LIN {X 0,Y 453.558,Z 377.477,A -85,B 0,C 180,E1 -8448.378,E2 -8448.378} C_VEL
LIN {X 0,Y 453.65,Z 377.467,A -85,B 0,C 180,E1 -8451.985,E2 -8451.985} C_VEL
LIN {X 0,Y 453.669,Z 377.47,A -85,B 0,C 180,E1 -8454.666,E2 -8454.666} C_VEL
LIN {X 0,Y 453.763,Z 377.461,A -85,B 0,C 180,E1 -8457.336,E2 -8457.336} C_VEL
LIN {X 0,Y 453.82,Z 377.435,A -85,B 0,C 180,E1 -8459.999,E2 -8459.999} C_VEL
LIN {X 0,Y 453.763,Z 377.452,A -85,B 0,C 180,E1 -8462.663,E2 -8462.663} C_VEL
LIN {X 0,Y 453.674,Z 377.469,A -85,B 0,C 180,E1 -8466.225,E2 -8466.225} C_VEL
LIN {X 0,Y 453.59,Z 377.471,A -85,B 0,C 180,E1 -8468.913,E2 -8468.913} C_VEL
LIN {X 0,Y 453.599,Z 377.475,A -85,B 0,C 180,E1 -8472.55,E2 -8472.55} C_VEL
LIN {X 0,Y 453.541,Z 377.484,A -85,B 0,C 180,E1 -8476.195,E2 -8476.195} C_VEL
LIN {X 0,Y 453.516,Z 377.479,A -85,B 0,C 180,E1 -8479.04,E2 -8479.04} C_VEL
LIN {X 0,Y 453.473,Z 377.497,A -85,B 0,C 180,E1 -8481.836,E2 -8481.836} C_VEL
LIN {X 0,Y 453.511,Z 377.49,A -85,B 0,C 180,E1 -8484.734,E2 -8484.734} C_VEL
LIN {X 0,Y 453.534,Z 377.482,A -85,B 0,C 180,E1 -8487.961,E2 -8487.961} C_VEL
LIN {X 0,Y 453.463,Z 377.502,A -85,B 0,C 180,E1 -8491.525,E2 -8491.525} C_VEL
LIN {X 0,Y 453.485,Z 377.484,A -85,B 0,C 180,E1 -8494.777,E2 -8494.777} C_VEL
LIN {X 0,Y 453.469,Z 377.496,A -85,B 0,C 180,E1 -8498.31,E2 -8498.31} C_VEL
LIN {X 0,Y 453.49,Z 377.486,A -85,B 0,C 180,E1 -8500.609,E2 -8500.609} C_VEL
LIN {X 0,Y 453.46,Z 377.502,A -85,B 0,C 180,E1 -8503.245,E2 -8503.245} C_VEL
LIN {X 0,Y 453.46,Z 377.488,A -85,B 0,C 180,E1 -8505.779,E2 -8505.779} C_VEL
LIN {X 0,Y 453.512,Z 377.477,A -85,B 0,C 180,E1 -8509.405,E2 -8509.405} C_VEL
LIN {X 0,Y 453.473,Z 377.496,A -85,B 0,C 180,E1 -8512.223,E2 -8512.223} C_VEL
LIN {X 0,Y 453.485,Z 377.482,A -85,B 0,C 180,E1 -8515.222,E2 -8515.222} C_VEL
LIN {X 0,Y 453.465,Z 377.498,A -85,B 0,C 180,E1 -8518.474,E2 -8518.474} C_VEL
LIN {X 0,Y 453.512,Z 377.486,A -85,B 0,C 180,E1 -8521.288,E2 -8521.288} C_VEL
LIN {X 0,Y 453.521,Z 377.491,A -85,B 0,C 180,E1 -8524.285,E2 -8524.285} C_VEL
LIN {X 0,Y 453.476,Z 377.501,A -85,B 0,C 180,E1 -8527.204,E2 -8527.204} C_VEL
LIN {X 0,Y 453.502,Z 377.494,A -85,B 0,C 180,E1 -8530.066,E2 -8530.066} C_VEL
LIN {X 0,Y 453.503,Z 377.497,A -85,B 0,C 180,E1 -8532.876,E2 -8532.876} C_VEL
LIN {X 0,Y 453.51,Z 377.495,A -85,B 0,C 180,E1 -8535.644,E2 -8535.644} C_VEL
LIN {X 0,Y 453.556,Z 377.489,A -85,B 0,C 180,E1 -8538.379,E2 -8538.379} C_VEL
LIN {X 0,Y 453.648,Z 377.477,A -85,B 0,C 180,E1 -8541.985,E2 -8541.985} C_VEL
LIN {X 0,Y 453.634,Z 377.48,A -85,B 0,C 180,E1 -8543.094,E2 -8543.094} C_VEL
LIN {X 0,Y 452.95,Z 377.564,A -85,B 0,C 180,E1 -8543.834,E2 -8543.834} C_VEL
LIN {X 0,Y 450.001,Z 377.934,A -85,B 0,C 180,E1 -8545.036,E2 -8545.036} C_VEL
LIN {X 0,Y 447.578,Z 378.234,A -85,B 0,C 180,E1 -8546.005,E2 -8546.005} C_VEL
LIN {X 0,Y 446.641,Z 378.352,A -85,B 0,C 180,E1 -8546.756,E2 -8546.756} C_VEL
LIN {X 0,Y 446.621,Z 378.353,A -85,B 0,C 180,E1 -8547.009,E2 -8547.009} C_VEL
LIN {X 0,Y 446.791,Z 378.332,A -85,B 0,C 180,E1 -8550,E2 -8550} C_VEL
LIN {X 0,Y 446.706,Z 378.344,A -85,B 0,C 180,E1 -8552.705,E2 -8552.705} C_VEL
LIN {X 0,Y 446.644,Z 378.35,A -85,B 0,C 180,E1 -8556.323,E2 -8556.323} C_VEL
LIN {X 0,Y 446.534,Z 378.366,A -85,B 0,C 180,E1 -8559.055,E2 -8559.055} C_VEL
LIN {X 0,Y 446.517,Z 378.368,A -85,B 0,C 180,E1 -8562.729,E2 -8562.729} C_VEL
LIN {X 0,Y 446.492,Z 378.368,A -85,B 0,C 180,E1 -8566.228,E2 -8566.228} C_VEL
LIN {X 0,Y 446.465,Z 378.373,A -85,B 0,C 180,E1 -8569.303,E2 -8569.303} C_VEL
LIN {X 0,Y 446.413,Z 378.378,A -85,B 0,C 180,E1 -8572.199,E2 -8572.199} C_VEL
LIN {X 0,Y 446.453,Z 378.375,A -85,B 0,C 180,E1 -8575.152,E2 -8575.152} C_VEL
LIN {X 0,Y 446.479,Z 378.368,A -85,B 0,C 180,E1 -8578.178,E2 -8578.178} C_VEL
LIN {X 0,Y 446.414,Z 378.378,A -85,B 0,C 180,E1 -8581.3,E2 -8581.3} C_VEL
LIN {X 0,Y 446.424,Z 378.361,A -85,B 0,C 180,E1 -8584.523,E2 -8584.523} C_VEL
LIN {X 0,Y 446.431,Z 378.374,A -85,B 0,C 180,E1 -8588.083,E2 -8588.083} C_VEL
LIN {X 0,Y 446.436,Z 378.353,A -85,B 0,C 180,E1 -8590.92,E2 -8590.92} C_VEL
LIN {X 0,Y 446.393,Z 378.365,A -85,B 0,C 180,E1 -8593.846,E2 -8593.846} C_VEL
LIN {X 0,Y 446.414,Z 378.378,A -85,B 0,C 180,E1 -8596.4,E2 -8596.4} C_VEL
LIN {X 0,Y 446.458,Z 378.362,A -85,B 0,C 180,E1 -8599.804,E2 -8599.804} C_VEL
LIN {X 0,Y 446.422,Z 378.376,A -85,B 0,C 180,E1 -8602.123,E2 -8602.123} C_VEL
LIN {X 0,Y 446.423,Z 378.362,A -85,B 0,C 180,E1 -8605.477,E2 -8605.477} C_VEL
LIN {X 0,Y 446.424,Z 378.379,A -85,B 0,C 180,E1 -8608.701,E2 -8608.701} C_VEL
LIN {X 0,Y 446.477,Z 378.359,A -85,B 0,C 180,E1 -8611.821,E2 -8611.821} C_VEL
LIN {X 0,Y 446.451,Z 378.372,A -85,B 0,C 180,E1 -8614.848,E2 -8614.848} C_VEL
LIN {X 0,Y 446.441,Z 378.374,A -85,B 0,C 180,E1 -8618.245,E2 -8618.245} C_VEL
LIN {X 0,Y 446.45,Z 378.357,A -85,B 0,C 180,E1 -8621.649,E2 -8621.649} C_VEL
LIN {X 0,Y 446.5,Z 378.369,A -85,B 0,C 180,E1 -8624.48,E2 -8624.48} C_VEL
LIN {X 0,Y 446.532,Z 378.356,A -85,B 0,C 180,E1 -8628.194,E2 -8628.194} C_VEL
LIN {X 0,Y 446.593,Z 378.343,A -85,B 0,C 180,E1 -8631.858,E2 -8631.858} C_VEL
LIN {X 0,Y 446.64,Z 378.351,A -85,B 0,C 180,E1 -8634.583,E2 -8634.583} C_VEL
LIN {X 0,Y 446.704,Z 378.331,A -85,B 0,C 180,E1 -8637.295,E2 -8637.295} C_VEL
LIN {X 0,Y 446.787,Z 378.31,A -85,B 0,C 180,E1 -8640.001,E2 -8640.001} C_VEL
LIN {X 0,Y 446.704,Z 378.34,A -85,B 0,C 180,E1 -8642.706,E2 -8642.706} C_VEL
LIN {X 0,Y 446.641,Z 378.347,A -85,B 0,C 180,E1 -8646.324,E2 -8646.324} C_VEL
LIN {X 0,Y 446.532,Z 378.339,A -85,B 0,C 180,E1 -8649.056,E2 -8649.056} C_VEL
LIN {X 0,Y 446.516,Z 378.362,A -85,B 0,C 180,E1 -8652.73,E2 -8652.73} C_VEL
LIN {X 0,Y 446.514,Z 378.359,A -85,B 0,C 180,E1 -8656.239,E2 -8656.239} C_VEL
LIN {X 0,Y 446.465,Z 378.354,A -85,B 0,C 180,E1 -8659.304,E2 -8659.304} C_VEL
LIN {X 0,Y 446.415,Z 378.379,A -85,B 0,C 180,E1 -8662.2,E2 -8662.2} C_VEL
LIN {X 0,Y 446.454,Z 378.362,A -85,B 0,C 180,E1 -8665.153,E2 -8665.153} C_VEL
LIN {X 0,Y 446.481,Z 378.362,A -85,B 0,C 180,E1 -8668.179,E2 -8668.179} C_VEL
LIN {X 0,Y 446.427,Z 378.372,A -85,B 0,C 180,E1 -8671.3,E2 -8671.3} C_VEL
LIN {X 0,Y 446.428,Z 378.369,A -85,B 0,C 180,E1 -8674.524,E2 -8674.524} C_VEL
LIN {X 0,Y 446.433,Z 378.376,A -85,B 0,C 180,E1 -8678.083,E2 -8678.083} C_VEL
LIN {X 0,Y 446.445,Z 378.369,A -85,B 0,C 180,E1 -8680.921,E2 -8680.921} C_VEL
LIN {X 0,Y 446.444,Z 378.373,A -85,B 0,C 180,E1 -8683.841,E2 -8683.841} C_VEL
LIN {X 0,Y 446.398,Z 378.379,A -85,B 0,C 180,E1 -8686.404,E2 -8686.404} C_VEL
LIN {X 0,Y 446.426,Z 378.36,A -85,B 0,C 180,E1 -8689.083,E2 -8689.083} C_VEL
LIN {X 0,Y 446.428,Z 378.377,A -85,B 0,C 180,E1 -8692.124,E2 -8692.124} C_VEL
LIN {X 0,Y 446.431,Z 378.374,A -85,B 0,C 180,E1 -8695.478,E2 -8695.478} C_VEL
LIN {X 0,Y 446.42,Z 378.379,A -85,B 0,C 180,E1 -8698.701,E2 -8698.701} C_VEL
LIN {X 0,Y 446.512,Z 378.494,A -85,B 0,C 180,E1 -8701.772,E2 -8701.772} C_VEL
LIN {X 0,Y 448.442,Z 388.8,A -85,B 0,C 180,E1 -8704.471,E2 -8704.471} C_VEL
LIN {X 0,Y 448.47,Z 393.611,A -85,B 0,C 180,E1 -8705.648,E2 -8705.648} C_VEL
LIN {X 0,Y 447.625,Z 408.364,A -85,B 0,C 180,E1 -8709.073,E2 -8709.073} C_VEL
LIN {X 0,Y 447.063,Z 419.525,A -85,B 0,C 180,E1 -8711.675,E2 -8711.675} C_VEL
LIN {X 0,Y 447.001,Z 421.52,A -85,B 0,C 180,E1 -8712.118,E2 -8712.118} C_VEL
LIN {X 0,Y 447.522,Z 425.001,A -85,B 0,C 180,E1 -8712.245,E2 -8712.245} C_VEL
LIN {X 0,Y 450.815,Z 444.234,A -85,B 0,C 180,E1 -8712.692,E2 -8712.692} C_VEL
LIN {X 0,Y 450.099,Z 526.468,A -85,B 0,C 180,E1 -8714.026,E2 -8714.026} C_VEL
LIN {X 0,Y 449.878,Z 536.383,A -85,B 0,C 180,E1 -8714.28,E2 -8714.28} C_VEL
LIN {X 0,Y 449.434,Z 546.367,A -85,B 0,C 180,E1 -8714.642,E2 -8714.642} C_VEL
LIN {X 0,Y 448.998,Z 556.725,A -85,B 0,C 180,E1 -8715.149,E2 -8715.149} C_VEL
LIN {X 0,Y 448.513,Z 565.872,A -85,B 0,C 180,E1 -8715.712,E2 -8715.712} C_VEL
LIN {X 0,Y 448.042,Z 574.876,A -85,B 0,C 180,E1 -8716.392,E2 -8716.392} C_VEL
LIN {X 0,Y 447.62,Z 583.474,A -85,B 0,C 180,E1 -8717.173,E2 -8717.173} C_VEL
LIN {X 0,Y 447.176,Z 591.031,A -85,B 0,C 180,E1 -8717.981,E2 -8717.981} C_VEL
LIN {X 0,Y 446.597,Z 599.827,A -85,B 0,C 180,E1 -8719.115,E2 -8719.115} C_VEL
LIN {X 0,Y 446.311,Z 605.819,A -85,B 0,C 180,E1 -8720.026,E2 -8720.026} C_VEL
LIN {X 0,Y 445.975,Z 612.13,A -85,B 0,C 180,E1 -8721.162,E2 -8721.162} C_VEL
LIN {X 0,Y 445.736,Z 617.404,A -85,B 0,C 180,E1 -8722.298,E2 -8722.298} C_VEL
LIN {X 0,Y 445.531,Z 622.495,A -85,B 0,C 180,E1 -8723.661,E2 -8723.661} C_VEL
LIN {X 0,Y 445.476,Z 626.458,A -85,B 0,C 180,E1 -8725.023,E2 -8725.023} C_VEL
LIN {X 0,Y 445.379,Z 629.387,A -85,B 0,C 180,E1 -8726.381,E2 -8726.381} C_VEL
LIN {X 0,Y 445.433,Z 630.887,A -85,B 0,C 180,E1 -8727.287,E2 -8727.287} C_VEL
LIN {X 0,Y 445.339,Z 632.404,A -85,B 0,C 180,E1 -8729.096,E2 -8729.096} C_VEL
LIN {X 0,Y 445.342,Z 632.682,A -85,B 0,C 180,E1 -8730,E2 -8730} C_VEL
LIN {X 0,Y 445.356,Z 631.81,A -85,B 0,C 180,E1 -8731.809,E2 -8731.809} C_VEL
LIN {X 0,Y 445.433,Z 630.886,A -85,B 0,C 180,E1 -8732.713,E2 -8732.713} C_VEL
LIN {X 0,Y 445.413,Z 627.543,A -85,B 0,C 180,E1 -8734.525,E2 -8734.525} C_VEL
LIN {X 0,Y 445.484,Z 625.333,A -85,B 0,C 180,E1 -8735.432,E2 -8735.432} C_VEL
LIN {X 0,Y 445.577,Z 621.153,A -85,B 0,C 180,E1 -8736.748,E2 -8736.748} C_VEL
LIN {X 0,Y 445.801,Z 615.405,A -85,B 0,C 180,E1 -8738.157,E2 -8738.157} C_VEL
LIN {X 0,Y 446.082,Z 609.751,A -85,B 0,C 180,E1 -8739.293,E2 -8739.293} C_VEL
LIN {X 0,Y 446.431,Z 602.945,A -85,B 0,C 180,E1 -8740.43,E2 -8740.43} C_VEL
LIN {X 0,Y 446.962,Z 594.728,A -85,B 0,C 180,E1 -8741.565,E2 -8741.565} C_VEL
LIN {X 0,Y 447.404,Z 586.898,A -85,B 0,C 180,E1 -8742.474,E2 -8742.474} C_VEL
LIN {X 0,Y 447.844,Z 579.107,A -85,B 0,C 180,E1 -8743.242,E2 -8743.242} C_VEL
LIN {X 0,Y 448.382,Z 569.046,A -85,B 0,C 180,E1 -8744.061,E2 -8744.061} C_VEL
LIN {X 0,Y 448.806,Z 560.653,A -85,B 0,C 180,E1 -8744.626,E2 -8744.626} C_VEL
LIN {X 0,Y 449.336,Z 550.145,A -85,B 0,C 180,E1 -8745.188,E2 -8745.188} C_VEL
LIN {X 0,Y 449.657,Z 539.808,A -85,B 0,C 180,E1 -8745.612,E2 -8745.612} C_VEL
LIN {X 0,Y 450.087,Z 529.088,A -85,B 0,C 180,E1 -8745.916,E2 -8745.916} C_VEL
LIN {X 0,Y 450.34,Z 505.147,A -85,B 0,C 180,E1 -8746.333,E2 -8746.333} C_VEL
LIN {X 0,Y 450.698,Z 443.314,A -85,B 0,C 180,E1 -8747.327,E2 -8747.327} C_VEL
LIN {X 0,Y 447.025,Z 421.937,A -85,B 0,C 180,E1 -8747.843,E2 -8747.843} C_VEL
LIN {X 0,Y 447.028,Z 420.542,A -85,B 0,C 180,E1 -8748.074,E2 -8748.074} C_VEL
LIN {X 0,Y 447.709,Z 407.508,A -85,B 0,C 180,E1 -8751.164,E2 -8751.164} C_VEL
LIN {X 0,Y 448.402,Z 395.093,A -85,B 0,C 180,E1 -8754.048,E2 -8754.048} C_VEL
LIN {X 0,Y 448.559,Z 389.849,A -85,B 0,C 180,E1 -8755.274,E2 -8755.274} C_VEL
LIN {X 0,Y 446.942,Z 380.625,A -85,B 0,C 180,E1 -8757.637,E2 -8757.637} C_VEL
LIN {X 0,Y 446.51,Z 378.449,A -85,B 0,C 180,E1 -8758.292,E2 -8758.292} C_VEL
LIN {X 0,Y 446.438,Z 378.376,A -85,B 0,C 180,E1 -8761.778,E2 -8761.778} C_VEL
LIN {X 0,Y 446.433,Z 378.372,A -85,B 0,C 180,E1 -8765.053,E2 -8765.053} C_VEL
LIN {X 0,Y 446.433,Z 378.379,A -85,B 0,C 180,E1 -8768.081,E2 -8768.081} C_VEL
LIN {X 0,Y 446.428,Z 378.359,A -85,B 0,C 180,E1 -8770.917,E2 -8770.917} C_VEL
LIN {X 0,Y 446.403,Z 378.381,A -85,B 0,C 180,E1 -8773.845,E2 -8773.845} C_VEL
LIN {X 0,Y 446.448,Z 378.372,A -85,B 0,C 180,E1 -8776.396,E2 -8776.396} C_VEL
LIN {X 0,Y 446.469,Z 378.367,A -85,B 0,C 180,E1 -8779.804,E2 -8779.804} C_VEL
LIN {X 0,Y 446.432,Z 378.377,A -85,B 0,C 180,E1 -8782.123,E2 -8782.123} C_VEL
LIN {X 0,Y 446.431,Z 378.369,A -85,B 0,C 180,E1 -8785.477,E2 -8785.477} C_VEL
LIN {X 0,Y 446.42,Z 378.373,A -85,B 0,C 180,E1 -8788.699,E2 -8788.699} C_VEL
LIN {X 0,Y 446.484,Z 378.362,A -85,B 0,C 180,E1 -8791.821,E2 -8791.821} C_VEL
LIN {X 0,Y 446.457,Z 378.362,A -85,B 0,C 180,E1 -8794.847,E2 -8794.847} C_VEL
LIN {X 0,Y 446.448,Z 378.369,A -85,B 0,C 180,E1 -8798.244,E2 -8798.244} C_VEL
LIN {X 0,Y 446.456,Z 378.356,A -85,B 0,C 180,E1 -8801.649,E2 -8801.649} C_VEL
LIN {X 0,Y 446.515,Z 378.359,A -85,B 0,C 180,E1 -8804.48,E2 -8804.48} C_VEL
LIN {X 0,Y 446.516,Z 378.355,A -85,B 0,C 180,E1 -8808.193,E2 -8808.193} C_VEL
LIN {X 0,Y 446.599,Z 378.341,A -85,B 0,C 180,E1 -8811.857,E2 -8811.857} C_VEL
LIN {X 0,Y 446.644,Z 378.345,A -85,B 0,C 180,E1 -8814.582,E2 -8814.582} C_VEL
LIN {X 0,Y 446.707,Z 378.339,A -85,B 0,C 180,E1 -8817.294,E2 -8817.294} C_VEL
LIN {X 0,Y 446.79,Z 378.31,A -85,B 0,C 180,E1 -8819.999,E2 -8819.999} C_VEL
LIN {X 0,Y 446.707,Z 378.331,A -85,B 0,C 180,E1 -8822.705,E2 -8822.705} C_VEL
LIN {X 0,Y 446.644,Z 378.344,A -85,B 0,C 180,E1 -8826.323,E2 -8826.323} C_VEL
LIN {X 0,Y 446.536,Z 378.351,A -85,B 0,C 180,E1 -8829.055,E2 -8829.055} C_VEL
LIN {X 0,Y 446.531,Z 378.355,A -85,B 0,C 180,E1 -8832.729,E2 -8832.729} C_VEL
LIN {X 0,Y 446.487,Z 378.362,A -85,B 0,C 180,E1 -8836.459,E2 -8836.459} C_VEL
LIN {X 0,Y 446.466,Z 378.356,A -85,B 0,C 180,E1 -8839.303,E2 -8839.303} C_VEL
LIN {X 0,Y 446.414,Z 378.374,A -85,B 0,C 180,E1 -8842.199,E2 -8842.199} C_VEL
LIN {X 0,Y 446.455,Z 378.372,A -85,B 0,C 180,E1 -8845.152,E2 -8845.152} C_VEL
LIN {X 0,Y 446.481,Z 378.359,A -85,B 0,C 180,E1 -8848.178,E2 -8848.178} C_VEL
LIN {X 0,Y 446.416,Z 378.376,A -85,B 0,C 180,E1 -8851.775,E2 -8851.775} C_VEL
LIN {X 0,Y 446.426,Z 378.362,A -85,B 0,C 180,E1 -8854.523,E2 -8854.523} C_VEL
LIN {X 0,Y 446.426,Z 378.374,A -85,B 0,C 180,E1 -8858.081,E2 -8858.081} C_VEL
LIN {X 0,Y 446.423,Z 378.368,A -85,B 0,C 180,E1 -8860.917,E2 -8860.917} C_VEL
LIN {X 0,Y 446.419,Z 378.375,A -85,B 0,C 180,E1 -8863.843,E2 -8863.843} C_VEL
LIN {X 0,Y 446.394,Z 378.365,A -85,B 0,C 180,E1 -8866.403,E2 -8866.403} C_VEL
LIN {X 0,Y 446.464,Z 378.363,A -85,B 0,C 180,E1 -8869.805,E2 -8869.805} C_VEL
LIN {X 0,Y 446.429,Z 378.374,A -85,B 0,C 180,E1 -8872.123,E2 -8872.123} C_VEL
LIN {X 0,Y 446.426,Z 378.361,A -85,B 0,C 180,E1 -8875.477,E2 -8875.477} C_VEL
LIN {X 0,Y 446.416,Z 378.377,A -85,B 0,C 180,E1 -8878.7,E2 -8878.7} C_VEL
LIN {X 0,Y 446.481,Z 378.368,A -85,B 0,C 180,E1 -8881.821,E2 -8881.821} C_VEL
LIN {X 0,Y 446.454,Z 378.375,A -85,B 0,C 180,E1 -8884.848,E2 -8884.848} C_VEL
LIN {X 0,Y 446.445,Z 378.373,A -85,B 0,C 180,E1 -8888.245,E2 -8888.245} C_VEL
LIN {X 0,Y 446.454,Z 378.374,A -85,B 0,C 180,E1 -8891.649,E2 -8891.649} C_VEL
LIN {X 0,Y 446.504,Z 378.367,A -85,B 0,C 180,E1 -8894.48,E2 -8894.48} C_VEL
LIN {X 0,Y 446.514,Z 378.366,A -85,B 0,C 180,E1 -8898.193,E2 -8898.193} C_VEL
LIN {X 0,Y 446.597,Z 378.356,A -85,B 0,C 180,E1 -8901.858,E2 -8901.858} C_VEL
LIN {X 0,Y 446.644,Z 378.352,A -85,B 0,C 180,E1 -8904.582,E2 -8904.582} C_VEL
LIN {X 0,Y 446.621,Z 378.353,A -85,B 0,C 180,E1 -8907.009,E2 -8907.009} C_VEL
LIN {X 0,Y 446.104,Z 378.421,A -85,B 0,C 180,E1 -8907.762,E2 -8907.762} C_VEL
LIN {X 0,Y 443.287,Z 378.776,A -85,B 0,C 180,E1 -8908.985,E2 -8908.985} C_VEL
LIN {X 0,Y 440.801,Z 379.085,A -85,B 0,C 180,E1 -8909.972,E2 -8909.972} C_VEL
LIN {X 0,Y 439.712,Z 379.217,A -85,B 0,C 180,E1 -8910.735,E2 -8910.735} C_VEL
LIN {X 0,Y 439.618,Z 379.226,A -85,B 0,C 180,E1 -8910.994,E2 -8910.994} C_VEL
LIN {X 0,Y 439.652,Z 379.222,A -85,B 0,C 180,E1 -8912.748,E2 -8912.748} C_VEL
LIN {X 0,Y 439.616,Z 379.227,A -85,B 0,C 180,E1 -8916.425,E2 -8916.425} C_VEL
LIN {X 0,Y 439.496,Z 379.242,A -85,B 0,C 180,E1 -8919.201,E2 -8919.201} C_VEL
LIN {X 0,Y 439.461,Z 379.247,A -85,B 0,C 180,E1 -8922.937,E2 -8922.937} C_VEL
LIN {X 0,Y 439.443,Z 379.247,A -85,B 0,C 180,E1 -8926.349,E2 -8926.349} C_VEL
LIN {X 0,Y 439.398,Z 379.252,A -85,B 0,C 180,E1 -8929.626,E2 -8929.626} C_VEL
LIN {X 0,Y 439.36,Z 379.259,A -85,B 0,C 180,E1 -8932.575,E2 -8932.575} C_VEL
LIN {X 0,Y 439.4,Z 379.251,A -85,B 0,C 180,E1 -8935.585,E2 -8935.585} C_VEL
LIN {X 0,Y 439.419,Z 379.24,A -85,B 0,C 180,E1 -8938.673,E2 -8938.673} C_VEL
LIN {X 0,Y 439.369,Z 379.254,A -85,B 0,C 180,E1 -8941.86,E2 -8941.86} C_VEL
LIN {X 0,Y 439.395,Z 379.238,A -85,B 0,C 180,E1 -8945.156,E2 -8945.156} C_VEL
LIN {X 0,Y 439.392,Z 379.255,A -85,B 0,C 180,E1 -8948.593,E2 -8948.593} C_VEL
LIN {X 0,Y 439.391,Z 379.226,A -85,B 0,C 180,E1 -8951.258,E2 -8951.258} C_VEL
LIN {X 0,Y 439.395,Z 379.246,A -85,B 0,C 180,E1 -8954.729,E2 -8954.729} C_VEL
LIN {X 0,Y 439.391,Z 379.248,A -85,B 0,C 180,E1 -8957.796,E2 -8957.796} C_VEL
LIN {X 0,Y 439.438,Z 379.239,A -85,B 0,C 180,E1 -8960.229,E2 -8960.229} C_VEL
LIN {X 0,Y 439.37,Z 379.25,A -85,B 0,C 180,E1 -8963.713,E2 -8963.713} C_VEL
LIN {X 0,Y 439.366,Z 379.253,A -85,B 0,C 180,E1 -8967.054,E2 -8967.054} C_VEL
LIN {X 0,Y 439.39,Z 379.253,A -85,B 0,C 180,E1 -8970.275,E2 -8970.275} C_VEL
LIN {X 0,Y 439.426,Z 379.236,A -85,B 0,C 180,E1 -8973.589,E2 -8973.589} C_VEL
LIN {X 0,Y 439.38,Z 379.256,A -85,B 0,C 180,E1 -8976.43,E2 -8976.43} C_VEL
LIN {X 0,Y 439.381,Z 379.241,A -85,B 0,C 180,E1 -8979.397,E2 -8979.397} C_VEL
LIN {X 0,Y 439.424,Z 379.237,A -85,B 0,C 180,E1 -8982.31,E2 -8982.31} C_VEL
LIN {X 0,Y 439.44,Z 379.243,A -85,B 0,C 180,E1 -8985.174,E2 -8985.174} C_VEL
LIN {X 0,Y 439.501,Z 379.233,A -85,B 0,C 180,E1 -8988.002,E2 -8988.002} C_VEL
LIN {X 0,Y 439.541,Z 379.221,A -85,B 0,C 180,E1 -8991.727,E2 -8991.727} C_VEL
LIN {X 0,Y 439.615,Z 379.227,A -85,B 0,C 180,E1 -8994.496,E2 -8994.496} C_VEL
LIN {X 0,Y 439.63,Z 379.211,A -85,B 0,C 180,E1 -8998.168,E2 -8998.168} C_VEL
LIN {X 0,Y 439.757,Z 379.185,A -85,B 0,C 180,E1 -9000.001,E2 -9000.001} C_VEL
LIN {X 0,Y 439.651,Z 379.218,A -85,B 0,C 180,E1 -9002.749,E2 -9002.749} C_VEL
LIN {X 0,Y 439.612,Z 379.22,A -85,B 0,C 180,E1 -9006.426,E2 -9006.426} C_VEL
LIN {X 0,Y 439.494,Z 379.215,A -85,B 0,C 180,E1 -9009.202,E2 -9009.202} C_VEL
LIN {X 0,Y 439.461,Z 379.239,A -85,B 0,C 180,E1 -9012.938,E2 -9012.938} C_VEL
LIN {X 0,Y 439.455,Z 379.236,A -85,B 0,C 180,E1 -9016.355,E2 -9016.355} C_VEL
LIN {X 0,Y 439.398,Z 379.235,A -85,B 0,C 180,E1 -9019.627,E2 -9019.627} C_VEL
LIN {X 0,Y 439.362,Z 379.254,A -85,B 0,C 180,E1 -9022.576,E2 -9022.576} C_VEL
LIN {X 0,Y 439.402,Z 379.242,A -85,B 0,C 180,E1 -9025.586,E2 -9025.586} C_VEL
LIN {X 0,Y 439.422,Z 379.245,A -85,B 0,C 180,E1 -9028.674,E2 -9028.674} C_VEL
LIN {X 0,Y 439.38,Z 379.253,A -85,B 0,C 180,E1 -9032.034,E2 -9032.034} C_VEL
LIN {X 0,Y 439.393,Z 379.244,A -85,B 0,C 180,E1 -9035.342,E2 -9035.342} C_VEL
LIN {X 0,Y 439.393,Z 379.246,A -85,B 0,C 180,E1 -9038.594,E2 -9038.594} C_VEL
LIN {X 0,Y 439.403,Z 379.246,A -85,B 0,C 180,E1 -9041.26,E2 -9041.26} C_VEL
LIN {X 0,Y 439.407,Z 379.247,A -85,B 0,C 180,E1 -9044.729,E2 -9044.729} C_VEL
LIN {X 0,Y 439.395,Z 379.248,A -85,B 0,C 180,E1 -9047.797,E2 -9047.797} C_VEL
LIN {X 0,Y 439.429,Z 379.239,A -85,B 0,C 180,E1 -9050.229,E2 -9050.229} C_VEL
LIN {X 0,Y 439.377,Z 379.247,A -85,B 0,C 180,E1 -9053.714,E2 -9053.714} C_VEL
LIN {X 0,Y 439.376,Z 379.249,A -85,B 0,C 180,E1 -9057.055,E2 -9057.055} C_VEL
LIN {X 0,Y 439.398,Z 379.25,A -85,B 0,C 180,E1 -9060.276,E2 -9060.276} C_VEL
LIN {X 0,Y 439.476,Z 379.419,A -85,B 0,C 180,E1 -9061.556,E2 -9061.556} C_VEL
LIN {X 0,Y 441.246,Z 388.657,A -85,B 0,C 180,E1 -9064.024,E2 -9064.024} C_VEL
LIN {X 0,Y 441.578,Z 392.932,A -85,B 0,C 180,E1 -9065.121,E2 -9065.121} C_VEL
LIN {X 0,Y 440.783,Z 407.16,A -85,B 0,C 180,E1 -9068.487,E2 -9068.487} C_VEL
LIN {X 0,Y 440.04,Z 420.288,A -85,B 0,C 180,E1 -9071.614,E2 -9071.614} C_VEL
LIN {X 0,Y 440.029,Z 421.615,A -85,B 0,C 180,E1 -9071.855,E2 -9071.855} C_VEL
LIN {X 0,Y 443.898,Z 444.095,A -85,B 0,C 180,E1 -9072.415,E2 -9072.415} C_VEL
LIN {X 0,Y 443.452,Z 511.516,A -85,B 0,C 180,E1 -9073.514,E2 -9073.514} C_VEL
LIN {X 0,Y 443.198,Z 530.238,A -85,B 0,C 180,E1 -9073.86,E2 -9073.86} C_VEL
LIN {X 0,Y 442.719,Z 543.644,A -85,B 0,C 180,E1 -9074.285,E2 -9074.285} C_VEL
LIN {X 0,Y 442.242,Z 554.562,A -85,B 0,C 180,E1 -9074.799,E2 -9074.799} C_VEL
LIN {X 0,Y 441.617,Z 565.676,A -85,B 0,C 180,E1 -9075.485,E2 -9075.485} C_VEL
LIN {X 0,Y 441.13,Z 574.681,A -85,B 0,C 180,E1 -9076.174,E2 -9076.174} C_VEL
LIN {X 0,Y 440.719,Z 582.808,A -85,B 0,C 180,E1 -9076.919,E2 -9076.919} C_VEL
LIN {X 0,Y 440.213,Z 590.835,A -85,B 0,C 180,E1 -9077.788,E2 -9077.788} C_VEL
LIN {X 0,Y 439.598,Z 599.631,A -85,B 0,C 180,E1 -9078.94,E2 -9078.94} C_VEL
LIN {X 0,Y 439.262,Z 605.623,A -85,B 0,C 180,E1 -9079.864,E2 -9079.864} C_VEL
LIN {X 0,Y 438.906,Z 611.934,A -85,B 0,C 180,E1 -9081.019,E2 -9081.019} C_VEL
LIN {X 0,Y 438.666,Z 617.208,A -85,B 0,C 180,E1 -9082.173,E2 -9082.173} C_VEL
LIN {X 0,Y 438.445,Z 622.525,A -85,B 0,C 180,E1 -9083.631,E2 -9083.631} C_VEL
LIN {X 0,Y 438.386,Z 626.262,A -85,B 0,C 180,E1 -9084.942,E2 -9084.942} C_VEL
LIN {X 0,Y 438.28,Z 629.192,A -85,B 0,C 180,E1 -9086.323,E2 -9086.323} C_VEL
LIN {X 0,Y 438.341,Z 630.692,A -85,B 0,C 180,E1 -9087.243,E2 -9087.243} C_VEL
LIN {X 0,Y 438.252,Z 632.209,A -85,B 0,C 180,E1 -9089.081,E2 -9089.081} C_VEL
LIN {X 0,Y 438.253,Z 632.487,A -85,B 0,C 180,E1 -9090,E2 -9090} C_VEL
LIN {X 0,Y 438.279,Z 631.615,A -85,B 0,C 180,E1 -9091.838,E2 -9091.838} C_VEL
LIN {X 0,Y 438.341,Z 630.691,A -85,B 0,C 180,E1 -9092.757,E2 -9092.757} C_VEL
LIN {X 0,Y 438.342,Z 627.348,A -85,B 0,C 180,E1 -9094.598,E2 -9094.598} C_VEL
LIN {X 0,Y 438.384,Z 625.137,A -85,B 0,C 180,E1 -9095.52,E2 -9095.52} C_VEL
LIN {X 0,Y 438.51,Z 620.784,A -85,B 0,C 180,E1 -9096.904,E2 -9096.904} C_VEL
LIN {X 0,Y 438.75,Z 615.209,A -85,B 0,C 180,E1 -9098.289,E2 -9098.289} C_VEL
LIN {X 0,Y 439.053,Z 609.556,A -85,B 0,C 180,E1 -9099.444,E2 -9099.444} C_VEL
LIN {X 0,Y 439.403,Z 602.749,A -85,B 0,C 180,E1 -9100.599,E2 -9100.599} C_VEL
LIN {X 0,Y 439.972,Z 594.532,A -85,B 0,C 180,E1 -9101.752,E2 -9101.752} C_VEL
LIN {X 0,Y 440.442,Z 586.702,A -85,B 0,C 180,E1 -9102.674,E2 -9102.674} C_VEL
LIN {X 0,Y 440.948,Z 578.055,A -85,B 0,C 180,E1 -9103.53,E2 -9103.53} C_VEL
LIN {X 0,Y 441.473,Z 568.85,A -85,B 0,C 180,E1 -9104.285,E2 -9104.285} C_VEL
LIN {X 0,Y 441.916,Z 560.457,A -85,B 0,C 180,E1 -9104.859,E2 -9104.859} C_VEL
LIN {X 0,Y 442.478,Z 549.95,A -85,B 0,C 180,E1 -9105.429,E2 -9105.429} C_VEL
LIN {X 0,Y 442.829,Z 539.613,A -85,B 0,C 180,E1 -9105.859,E2 -9105.859} C_VEL
LIN {X 0,Y 443.27,Z 528.893,A -85,B 0,C 180,E1 -9106.168,E2 -9106.168} C_VEL
LIN {X 0,Y 443.542,Z 505.013,A -85,B 0,C 180,E1 -9106.59,E2 -9106.59} C_VEL
LIN {X 0,Y 443.899,Z 444.061,A -85,B 0,C 180,E1 -9107.586,E2 -9107.586} C_VEL
LIN {X 0,Y 440.035,Z 421.693,A -85,B 0,C 180,E1 -9108.14,E2 -9108.14} C_VEL
LIN {X 0,Y 440.019,Z 420.945,A -85,B 0,C 180,E1 -9108.231,E2 -9108.231} C_VEL
LIN {X 0,Y 440.783,Z 407.344,A -85,B 0,C 180,E1 -9111.513,E2 -9111.513} C_VEL
LIN {X 0,Y 441.519,Z 394.955,A -85,B 0,C 180,E1 -9114.448,E2 -9114.448} C_VEL
LIN {X 0,Y 441.569,Z 390.757,A -85,B 0,C 180,E1 -9115.45,E2 -9115.45} C_VEL
LIN {X 0,Y 439.77,Z 380.996,A -85,B 0,C 180,E1 -9118.001,E2 -9118.001} C_VEL
LIN {X 0,Y 439.467,Z 379.348,A -85,B 0,C 180,E1 -9118.493,E2 -9118.493} C_VEL
LIN {X 0,Y 439.389,Z 379.253,A -85,B 0,C 180,E1 -9121.859,E2 -9121.859} C_VEL
LIN {X 0,Y 439.404,Z 379.248,A -85,B 0,C 180,E1 -9125.155,E2 -9125.155} C_VEL
LIN {X 0,Y 439.391,Z 379.25,A -85,B 0,C 180,E1 -9128.594,E2 -9128.594} C_VEL
LIN {X 0,Y 439.39,Z 379.236,A -85,B 0,C 180,E1 -9131.256,E2 -9131.256} C_VEL
LIN {X 0,Y 439.404,Z 379.246,A -85,B 0,C 180,E1 -9134.729,E2 -9134.729} C_VEL
LIN {X 0,Y 439.414,Z 379.252,A -85,B 0,C 180,E1 -9137.797,E2 -9137.797} C_VEL
LIN {X 0,Y 439.45,Z 379.24,A -85,B 0,C 180,E1 -9140.229,E2 -9140.229} C_VEL
LIN {X 0,Y 439.377,Z 379.256,A -85,B 0,C 180,E1 -9143.713,E2 -9143.713} C_VEL
LIN {X 0,Y 439.376,Z 379.244,A -85,B 0,C 180,E1 -9147.054,E2 -9147.054} C_VEL
LIN {X 0,Y 439.397,Z 379.249,A -85,B 0,C 180,E1 -9150.275,E2 -9150.275} C_VEL
LIN {X 0,Y 439.433,Z 379.233,A -85,B 0,C 180,E1 -9153.588,E2 -9153.588} C_VEL
LIN {X 0,Y 439.387,Z 379.249,A -85,B 0,C 180,E1 -9156.429,E2 -9156.429} C_VEL
LIN {X 0,Y 439.388,Z 379.248,A -85,B 0,C 180,E1 -9159.397,E2 -9159.397} C_VEL
LIN {X 0,Y 439.431,Z 379.234,A -85,B 0,C 180,E1 -9162.309,E2 -9162.309} C_VEL
LIN {X 0,Y 439.451,Z 379.24,A -85,B 0,C 180,E1 -9165.174,E2 -9165.174} C_VEL
LIN {X 0,Y 439.482,Z 379.233,A -85,B 0,C 180,E1 -9168.001,E2 -9168.001} C_VEL
LIN {X 0,Y 439.546,Z 379.216,A -85,B 0,C 180,E1 -9171.726,E2 -9171.726} C_VEL
LIN {X 0,Y 439.619,Z 379.22,A -85,B 0,C 180,E1 -9174.495,E2 -9174.495} C_VEL
LIN {X 0,Y 439.634,Z 379.211,A -85,B 0,C 180,E1 -9178.167,E2 -9178.167} C_VEL
LIN {X 0,Y 439.76,Z 379.185,A -85,B 0,C 180,E1 -9179.999,E2 -9179.999} C_VEL
LIN {X 0,Y 439.654,Z 379.21,A -85,B 0,C 180,E1 -9182.748,E2 -9182.748} C_VEL
LIN {X 0,Y 439.615,Z 379.219,A -85,B 0,C 180,E1 -9186.425,E2 -9186.425} C_VEL
LIN {X 0,Y 439.498,Z 379.226,A -85,B 0,C 180,E1 -9189.201,E2 -9189.201} C_VEL
LIN {X 0,Y 439.501,Z 379.231,A -85,B 0,C 180,E1 -9192.726,E2 -9192.726} C_VEL
LIN {X 0,Y 439.444,Z 379.24,A -85,B 0,C 180,E1 -9196.348,E2 -9196.348} C_VEL
LIN {X 0,Y 439.399,Z 379.237,A -85,B 0,C 180,E1 -9199.626,E2 -9199.626} C_VEL
LIN {X 0,Y 439.361,Z 379.252,A -85,B 0,C 180,E1 -9202.575,E2 -9202.575} C_VEL
LIN {X 0,Y 439.402,Z 379.245,A -85,B 0,C 180,E1 -9205.584,E2 -9205.584} C_VEL
LIN {X 0,Y 439.414,Z 379.239,A -85,B 0,C 180,E1 -9208.673,E2 -9208.673} C_VEL
LIN {X 0,Y 439.367,Z 379.252,A -85,B 0,C 180,E1 -9212.03,E2 -9212.03} C_VEL
LIN {X 0,Y 439.392,Z 379.244,A -85,B 0,C 180,E1 -9215.34,E2 -9215.34} C_VEL
LIN {X 0,Y 439.384,Z 379.251,A -85,B 0,C 180,E1 -9218.594,E2 -9218.594} C_VEL
LIN {X 0,Y 439.385,Z 379.246,A -85,B 0,C 180,E1 -9221.257,E2 -9221.257} C_VEL
LIN {X 0,Y 439.401,Z 379.248,A -85,B 0,C 180,E1 -9224.728,E2 -9224.728} C_VEL
LIN {X 0,Y 439.393,Z 379.223,A -85,B 0,C 180,E1 -9227.796,E2 -9227.796} C_VEL
LIN {X 0,Y 439.446,Z 379.238,A -85,B 0,C 180,E1 -9230.23,E2 -9230.23} C_VEL
LIN {X 0,Y 439.373,Z 379.246,A -85,B 0,C 180,E1 -9233.713,E2 -9233.713} C_VEL
LIN {X 0,Y 439.369,Z 379.249,A -85,B 0,C 180,E1 -9237.054,E2 -9237.054} C_VEL
LIN {X 0,Y 439.393,Z 379.241,A -85,B 0,C 180,E1 -9240.275,E2 -9240.275} C_VEL
LIN {X 0,Y 439.43,Z 379.249,A -85,B 0,C 180,E1 -9243.588,E2 -9243.588} C_VEL
LIN {X 0,Y 439.383,Z 379.253,A -85,B 0,C 180,E1 -9246.429,E2 -9246.429} C_VEL
LIN {X 0,Y 439.386,Z 379.256,A -85,B 0,C 180,E1 -9249.397,E2 -9249.397} C_VEL
LIN {X 0,Y 439.428,Z 379.248,A -85,B 0,C 180,E1 -9252.309,E2 -9252.309} C_VEL
LIN {X 0,Y 439.444,Z 379.249,A -85,B 0,C 180,E1 -9255.174,E2 -9255.174} C_VEL
LIN {X 0,Y 439.48,Z 379.242,A -85,B 0,C 180,E1 -9258.001,E2 -9258.001} C_VEL
LIN {X 0,Y 439.544,Z 379.235,A -85,B 0,C 180,E1 -9261.726,E2 -9261.726} C_VEL
LIN {X 0,Y 439.619,Z 379.226,A -85,B 0,C 180,E1 -9264.496,E2 -9264.496} C_VEL
LIN {X 0,Y 439.632,Z 379.223,A -85,B 0,C 180,E1 -9268.168,E2 -9268.168} C_VEL
LIN {X 0,Y 439.761,Z 379.208,A -85,B 0,C 180,E1 -9270,E2 -9270} C_VEL
LIN {X 0,Y 439.618,Z 379.226,A -85,B 0,C 180,E1 -9270.994,E2 -9270.994} C_VEL
LIN {X 0,Y 438.902,Z 379.314,A -85,B 0,C 180,E1 -9271.758,E2 -9271.758} C_VEL
LIN {X 0,Y 435.924,Z 379.687,A -85,B 0,C 180,E1 -9272.997,E2 -9272.997} C_VEL
LIN {X 0,Y 433.473,Z 379.993,A -85,B 0,C 180,E1 -9273.998,E2 -9273.998} C_VEL
LIN {X 0,Y 432.5,Z 380.114,A -85,B 0,C 180,E1 -9274.772,E2 -9274.772} C_VEL
LIN {X 0,Y 432.463,Z 380.116,A -85,B 0,C 180,E1 -9275.034,E2 -9275.034} C_VEL
LIN {X 0,Y 432.582,Z 380.103,A -85,B 0,C 180,E1 -9277.679,E2 -9277.679} C_VEL
LIN {X 0,Y 432.389,Z 380.127,A -85,B 0,C 180,E1 -9281.247,E2 -9281.247} C_VEL
LIN {X 0,Y 432.369,Z 380.128,A -85,B 0,C 180,E1 -9284.112,E2 -9284.112} C_VEL
LIN {X 0,Y 432.393,Z 380.127,A -85,B 0,C 180,E1 -9287.011,E2 -9287.011} C_VEL
LIN {X 0,Y 432.334,Z 380.132,A -85,B 0,C 180,E1 -9289.96,E2 -9289.96} C_VEL
LIN {X 0,Y 432.314,Z 380.137,A -85,B 0,C 180,E1 -9292.964,E2 -9292.964} C_VEL
LIN {X 0,Y 432.359,Z 380.128,A -85,B 0,C 180,E1 -9296.032,E2 -9296.032} C_VEL
LIN {X 0,Y 432.347,Z 380.117,A -85,B 0,C 180,E1 -9299.186,E2 -9299.186} C_VEL
LIN {X 0,Y 432.32,Z 380.134,A -85,B 0,C 180,E1 -9302.293,E2 -9302.293} C_VEL
LIN {X 0,Y 432.335,Z 380.114,A -85,B 0,C 180,E1 -9304.677,E2 -9304.677} C_VEL
LIN {X 0,Y 432.346,Z 380.13,A -85,B 0,C 180,E1 -9308.148,E2 -9308.148} C_VEL
LIN {X 0,Y 432.36,Z 380.099,A -85,B 0,C 180,E1 -9311.607,E2 -9311.607} C_VEL
LIN {X 0,Y 432.326,Z 380.12,A -85,B 0,C 180,E1 -9314.347,E2 -9314.347} C_VEL
LIN {X 0,Y 432.318,Z 380.132,A -85,B 0,C 180,E1 -9317.015,E2 -9317.015} C_VEL
LIN {X 0,Y 432.345,Z 380.119,A -85,B 0,C 180,E1 -9319.818,E2 -9319.818} C_VEL
LIN {X 0,Y 432.309,Z 380.132,A -85,B 0,C 180,E1 -9323.023,E2 -9323.023} C_VEL
LIN {X 0,Y 432.352,Z 380.116,A -85,B 0,C 180,E1 -9325.996,E2 -9325.996} C_VEL
LIN {X 0,Y 432.388,Z 380.122,A -85,B 0,C 180,E1 -9329.744,E2 -9329.744} C_VEL
LIN {X 0,Y 432.393,Z 380.112,A -85,B 0,C 180,E1 -9333.372,E2 -9333.372} C_VEL
LIN {X 0,Y 432.364,Z 380.125,A -85,B 0,C 180,E1 -9336.024,E2 -9336.024} C_VEL
LIN {X 0,Y 432.343,Z 380.119,A -85,B 0,C 180,E1 -9339.046,E2 -9339.046} C_VEL
LIN {X 0,Y 432.371,Z 380.112,A -85,B 0,C 180,E1 -9342.011,E2 -9342.011} C_VEL
LIN {X 0,Y 432.388,Z 380.124,A -85,B 0,C 180,E1 -9344.927,E2 -9344.927} C_VEL
LIN {X 0,Y 432.474,Z 380.107,A -85,B 0,C 180,E1 -9347.804,E2 -9347.804} C_VEL
LIN {X 0,Y 432.485,Z 380.099,A -85,B 0,C 180,E1 -9351.591,E2 -9351.591} C_VEL
LIN {X 0,Y 432.592,Z 380.102,A -85,B 0,C 180,E1 -9354.407,E2 -9354.407} C_VEL
LIN {X 0,Y 432.6,Z 380.086,A -85,B 0,C 180,E1 -9358.139,E2 -9358.139} C_VEL
LIN {X 0,Y 432.727,Z 380.06,A -85,B 0,C 180,E1 -9360.001,E2 -9360.001} C_VEL
LIN {X 0,Y 432.6,Z 380.096,A -85,B 0,C 180,E1 -9362.794,E2 -9362.794} C_VEL
LIN {X 0,Y 432.567,Z 380.096,A -85,B 0,C 180,E1 -9366.531,E2 -9366.531} C_VEL
LIN {X 0,Y 432.437,Z 380.093,A -85,B 0,C 180,E1 -9369.354,E2 -9369.354} C_VEL
LIN {X 0,Y 432.426,Z 380.116,A -85,B 0,C 180,E1 -9372.804,E2 -9372.804} C_VEL
LIN {X 0,Y 432.418,Z 380.11,A -85,B 0,C 180,E1 -9376.484,E2 -9376.484} C_VEL
LIN {X 0,Y 432.334,Z 380.118,A -85,B 0,C 180,E1 -9379.961,E2 -9379.961} C_VEL
LIN {X 0,Y 432.315,Z 380.13,A -85,B 0,C 180,E1 -9382.965,E2 -9382.965} C_VEL
LIN {X 0,Y 432.361,Z 380.116,A -85,B 0,C 180,E1 -9386.033,E2 -9386.033} C_VEL
LIN {X 0,Y 432.349,Z 380.124,A -85,B 0,C 180,E1 -9389.188,E2 -9389.188} C_VEL
LIN {X 0,Y 432.329,Z 380.127,A -85,B 0,C 180,E1 -9392.295,E2 -9392.295} C_VEL
LIN {X 0,Y 432.338,Z 380.124,A -85,B 0,C 180,E1 -9394.678,E2 -9394.678} C_VEL
LIN {X 0,Y 432.349,Z 380.129,A -85,B 0,C 180,E1 -9398.149,E2 -9398.149} C_VEL
LIN {X 0,Y 432.371,Z 380.124,A -85,B 0,C 180,E1 -9401.609,E2 -9401.609} C_VEL
LIN {X 0,Y 432.377,Z 380.123,A -85,B 0,C 180,E1 -9404.342,E2 -9404.342} C_VEL
LIN {X 0,Y 432.332,Z 380.12,A -85,B 0,C 180,E1 -9408.204,E2 -9408.204} C_VEL
LIN {X 0,Y 432.35,Z 380.126,A -85,B 0,C 180,E1 -9411.285,E2 -9411.285} C_VEL
LIN {X 0,Y 432.346,Z 380.123,A -85,B 0,C 180,E1 -9414.369,E2 -9414.369} C_VEL
LIN {X 0,Y 432.328,Z 380.127,A -85,B 0,C 180,E1 -9417.558,E2 -9417.558} C_VEL
LIN {X 0,Y 432.363,Z 380.131,A -85,B 0,C 180,E1 -9420.815,E2 -9420.815} C_VEL
LIN {X 0,Y 432.464,Z 380.383,A -85,B 0,C 180,E1 -9421.35,E2 -9421.35} C_VEL
LIN {X 0,Y 434.359,Z 390.465,A -85,B 0,C 180,E1 -9424.097,E2 -9424.097} C_VEL
LIN {X 0,Y 434.59,Z 394.557,A -85,B 0,C 180,E1 -9425.137,E2 -9425.137} C_VEL
LIN {X 0,Y 433.814,Z 408.023,A -85,B 0,C 180,E1 -9428.374,E2 -9428.374} C_VEL
LIN {X 0,Y 433.028,Z 421.133,A -85,B 0,C 180,E1 -9431.52,E2 -9431.52} C_VEL
LIN {X 0,Y 433.553,Z 424.297,A -85,B 0,C 180,E1 -9431.648,E2 -9431.648} C_VEL
LIN {X 0,Y 437.22,Z 445.539,A -85,B 0,C 180,E1 -9432.165,E2 -9432.165} C_VEL
LIN {X 0,Y 436.483,Z 526.079,A -85,B 0,C 180,E1 -9433.514,E2 -9433.514} C_VEL
LIN {X 0,Y 436.242,Z 535.994,A -85,B 0,C 180,E1 -9433.775,E2 -9433.775} C_VEL
LIN {X 0,Y 435.761,Z 545.977,A -85,B 0,C 180,E1 -9434.148,E2 -9434.148} C_VEL
LIN {X 0,Y 435.258,Z 556.334,A -85,B 0,C 180,E1 -9434.669,E2 -9434.669} C_VEL
LIN {X 0,Y 434.75,Z 565.481,A -85,B 0,C 180,E1 -9435.25,E2 -9435.25} C_VEL
LIN {X 0,Y 434.217,Z 574.485,A -85,B 0,C 180,E1 -9435.95,E2 -9435.95} C_VEL
LIN {X 0,Y 433.745,Z 582.99,A -85,B 0,C 180,E1 -9436.745,E2 -9436.745} C_VEL
LIN {X 0,Y 433.252,Z 590.639,A -85,B 0,C 180,E1 -9437.589,E2 -9437.589} C_VEL
LIN {X 0,Y 432.614,Z 599.435,A -85,B 0,C 180,E1 -9438.759,E2 -9438.759} C_VEL
LIN {X 0,Y 432.226,Z 605.426,A -85,B 0,C 180,E1 -9439.697,E2 -9439.697} C_VEL
LIN {X 0,Y 431.854,Z 611.738,A -85,B 0,C 180,E1 -9440.871,E2 -9440.871} C_VEL
LIN {X 0,Y 431.59,Z 617.012,A -85,B 0,C 180,E1 -9442.044,E2 -9442.044} C_VEL
LIN {X 0,Y 431.378,Z 622.104,A -85,B 0,C 180,E1 -9443.452,E2 -9443.452} C_VEL
LIN {X 0,Y 431.297,Z 626.067,A -85,B 0,C 180,E1 -9444.858,E2 -9444.858} C_VEL
LIN {X 0,Y 431.187,Z 628.996,A -85,B 0,C 180,E1 -9446.262,E2 -9446.262} C_VEL
LIN {X 0,Y 431.236,Z 630.496,A -85,B 0,C 180,E1 -9447.198,E2 -9447.198} C_VEL
LIN {X 0,Y 431.169,Z 632.014,A -85,B 0,C 180,E1 -9449.066,E2 -9449.066} C_VEL
LIN {X 0,Y 431.167,Z 632.293,A -85,B 0,C 180,E1 -9450,E2 -9450} C_VEL
LIN {X 0,Y 431.203,Z 631.421,A -85,B 0,C 180,E1 -9451.868,E2 -9451.868} C_VEL
LIN {X 0,Y 431.236,Z 630.495,A -85,B 0,C 180,E1 -9452.803,E2 -9452.803} C_VEL
LIN {X 0,Y 431.272,Z 627.153,A -85,B 0,C 180,E1 -9454.674,E2 -9454.674} C_VEL
LIN {X 0,Y 431.287,Z 623.827,A -85,B 0,C 180,E1 -9455.982,E2 -9455.982} C_VEL
LIN {X 0,Y 431.431,Z 620.588,A -85,B 0,C 180,E1 -9457.018,E2 -9457.018} C_VEL
LIN {X 0,Y 431.69,Z 615.013,A -85,B 0,C 180,E1 -9458.426,E2 -9458.426} C_VEL
LIN {X 0,Y 432,Z 609.359,A -85,B 0,C 180,E1 -9459.599,E2 -9459.599} C_VEL
LIN {X 0,Y 432.398,Z 602.553,A -85,B 0,C 180,E1 -9460.773,E2 -9460.773} C_VEL
LIN {X 0,Y 432.984,Z 594.336,A -85,B 0,C 180,E1 -9461.944,E2 -9461.944} C_VEL
LIN {X 0,Y 433.474,Z 586.506,A -85,B 0,C 180,E1 -9462.881,E2 -9462.881} C_VEL
LIN {X 0,Y 434.009,Z 577.975,A -85,B 0,C 180,E1 -9463.74,E2 -9463.74} C_VEL
LIN {X 0,Y 434.565,Z 568.655,A -85,B 0,C 180,E1 -9464.517,E2 -9464.517} C_VEL
LIN {X 0,Y 435.048,Z 560.262,A -85,B 0,C 180,E1 -9465.099,E2 -9465.099} C_VEL
LIN {X 0,Y 435.625,Z 549.755,A -85,B 0,C 180,E1 -9465.678,E2 -9465.678} C_VEL
LIN {X 0,Y 436.015,Z 539.418,A -85,B 0,C 180,E1 -9466.114,E2 -9466.114} C_VEL
LIN {X 0,Y 436.463,Z 528.698,A -85,B 0,C 180,E1 -9466.427,E2 -9466.427} C_VEL
LIN {X 0,Y 436.755,Z 504.869,A -85,B 0,C 180,E1 -9466.854,E2 -9466.854} C_VEL
LIN {X 0,Y 437.162,Z 445.091,A -85,B 0,C 180,E1 -9467.845,E2 -9467.845} C_VEL
LIN {X 0,Y 433.102,Z 421.769,A -85,B 0,C 180,E1 -9468.425,E2 -9468.425} C_VEL
LIN {X 0,Y 433.042,Z 420.533,A -85,B 0,C 180,E1 -9468.582,E2 -9468.582} C_VEL
LIN {X 0,Y 433.851,Z 407.179,A -85,B 0,C 180,E1 -9471.875,E2 -9471.875} C_VEL
LIN {X 0,Y 434.717,Z 393.693,A -85,B 0,C 180,E1 -9475.13,E2 -9475.13} C_VEL
LIN {X 0,Y 434.007,Z 388.57,A -85,B 0,C 180,E1 -9476.428,E2 -9476.428} C_VEL
LIN {X 0,Y 432.436,Z 380.219,A -85,B 0,C 180,E1 -9478.745,E2 -9478.745} C_VEL
LIN {X 0,Y 432.333,Z 380.134,A -85,B 0,C 180,E1 -9481.345,E2 -9481.345} C_VEL
LIN {X 0,Y 432.344,Z 380.128,A -85,B 0,C 180,E1 -9484.677,E2 -9484.677} C_VEL
LIN {X 0,Y 432.349,Z 380.132,A -85,B 0,C 180,E1 -9488.148,E2 -9488.148} C_VEL
LIN {X 0,Y 432.334,Z 380.117,A -85,B 0,C 180,E1 -9491.601,E2 -9491.601} C_VEL
LIN {X 0,Y 432.335,Z 380.13,A -85,B 0,C 180,E1 -9494.347,E2 -9494.347} C_VEL
LIN {X 0,Y 432.367,Z 380.124,A -85,B 0,C 180,E1 -9497.009,E2 -9497.009} C_VEL
LIN {X 0,Y 432.358,Z 380.124,A -85,B 0,C 180,E1 -9499.817,E2 -9499.817} C_VEL
LIN {X 0,Y 432.317,Z 380.131,A -85,B 0,C 180,E1 -9503.022,E2 -9503.022} C_VEL
LIN {X 0,Y 432.36,Z 380.118,A -85,B 0,C 180,E1 -9505.996,E2 -9505.996} C_VEL
LIN {X 0,Y 432.395,Z 380.126,A -85,B 0,C 180,E1 -9509.744,E2 -9509.744} C_VEL
LIN {X 0,Y 432.4,Z 380.107,A -85,B 0,C 180,E1 -9513.372,E2 -9513.372} C_VEL
LIN {X 0,Y 432.371,Z 380.127,A -85,B 0,C 180,E1 -9516.023,E2 -9516.023} C_VEL
LIN {X 0,Y 432.35,Z 380.123,A -85,B 0,C 180,E1 -9519.046,E2 -9519.046} C_VEL
LIN {X 0,Y 432.377,Z 380.11,A -85,B 0,C 180,E1 -9522.011,E2 -9522.011} C_VEL
LIN {X 0,Y 432.401,Z 380.117,A -85,B 0,C 180,E1 -9524.926,E2 -9524.926} C_VEL
LIN {X 0,Y 432.458,Z 380.11,A -85,B 0,C 180,E1 -9527.803,E2 -9527.803} C_VEL
LIN {X 0,Y 432.49,Z 380.092,A -85,B 0,C 180,E1 -9531.59,E2 -9531.59} C_VEL
LIN {X 0,Y 432.596,Z 380.095,A -85,B 0,C 180,E1 -9534.406,E2 -9534.406} C_VEL
LIN {X 0,Y 432.604,Z 380.087,A -85,B 0,C 180,E1 -9538.138,E2 -9538.138} C_VEL
LIN {X 0,Y 432.729,Z 380.06,A -85,B 0,C 180,E1 -9539.999,E2 -9539.999} C_VEL
LIN {X 0,Y 432.603,Z 380.088,A -85,B 0,C 180,E1 -9542.793,E2 -9542.793} C_VEL
LIN {X 0,Y 432.57,Z 380.097,A -85,B 0,C 180,E1 -9546.53,E2 -9546.53} C_VEL
LIN {X 0,Y 432.441,Z 380.102,A -85,B 0,C 180,E1 -9549.353,E2 -9549.353} C_VEL
LIN {X 0,Y 432.442,Z 380.11,A -85,B 0,C 180,E1 -9552.811,E2 -9552.811} C_VEL
LIN {X 0,Y 432.409,Z 380.116,A -85,B 0,C 180,E1 -9556.478,E2 -9556.478} C_VEL
LIN {X 0,Y 432.335,Z 380.119,A -85,B 0,C 180,E1 -9559.96,E2 -9559.96} C_VEL
LIN {X 0,Y 432.316,Z 380.131,A -85,B 0,C 180,E1 -9562.964,E2 -9562.964} C_VEL
LIN {X 0,Y 432.361,Z 380.117,A -85,B 0,C 180,E1 -9566.032,E2 -9566.032} C_VEL
LIN {X 0,Y 432.339,Z 380.124,A -85,B 0,C 180,E1 -9569.187,E2 -9569.187} C_VEL
LIN {X 0,Y 432.319,Z 380.129,A -85,B 0,C 180,E1 -9572.443,E2 -9572.443} C_VEL
LIN {X 0,Y 432.341,Z 380.126,A -85,B 0,C 180,E1 -9575.632,E2 -9575.632} C_VEL
LIN {X 0,Y 432.347,Z 380.128,A -85,B 0,C 180,E1 -9578.716,E2 -9578.716} C_VEL
LIN {X 0,Y 432.331,Z 380.13,A -85,B 0,C 180,E1 -9581.797,E2 -9581.797} C_VEL
LIN {X 0,Y 432.336,Z 380.127,A -85,B 0,C 180,E1 -9584.346,E2 -9584.346} C_VEL
LIN {X 0,Y 432.316,Z 380.11,A -85,B 0,C 180,E1 -9587.015,E2 -9587.015} C_VEL
LIN {X 0,Y 432.352,Z 380.119,A -85,B 0,C 180,E1 -9589.817,E2 -9589.817} C_VEL
LIN {X 0,Y 432.313,Z 380.135,A -85,B 0,C 180,E1 -9593.023,E2 -9593.023} C_VEL
LIN {X 0,Y 432.356,Z 380.115,A -85,B 0,C 180,E1 -9595.996,E2 -9595.996} C_VEL
LIN {X 0,Y 432.391,Z 380.115,A -85,B 0,C 180,E1 -9599.744,E2 -9599.744} C_VEL
LIN {X 0,Y 432.396,Z 380.127,A -85,B 0,C 180,E1 -9603.372,E2 -9603.372} C_VEL
LIN {X 0,Y 432.368,Z 380.127,A -85,B 0,C 180,E1 -9606.023,E2 -9606.023} C_VEL
LIN {X 0,Y 432.347,Z 380.133,A -85,B 0,C 180,E1 -9609.046,E2 -9609.046} C_VEL
LIN {X 0,Y 432.375,Z 380.127,A -85,B 0,C 180,E1 -9612.011,E2 -9612.011} C_VEL
LIN {X 0,Y 432.392,Z 380.127,A -85,B 0,C 180,E1 -9614.926,E2 -9614.926} C_VEL
LIN {X 0,Y 432.456,Z 380.118,A -85,B 0,C 180,E1 -9617.803,E2 -9617.803} C_VEL
LIN {X 0,Y 432.488,Z 380.114,A -85,B 0,C 180,E1 -9621.59,E2 -9621.59} C_VEL
LIN {X 0,Y 432.596,Z 380.101,A -85,B 0,C 180,E1 -9624.406,E2 -9624.406} C_VEL
LIN {X 0,Y 432.602,Z 380.099,A -85,B 0,C 180,E1 -9628.138,E2 -9628.138} C_VEL
LIN {X 0,Y 432.73,Z 380.084,A -85,B 0,C 180,E1 -9630,E2 -9630} C_VEL
LIN {X 0,Y 432.602,Z 380.1,A -85,B 0,C 180,E1 -9632.793,E2 -9632.793} C_VEL
LIN {X 0,Y 432.463,Z 380.116,A -85,B 0,C 180,E1 -9635.034,E2 -9635.034} C_VEL
LIN {X 0,Y 431.904,Z 380.187,A -85,B 0,C 180,E1 -9635.813,E2 -9635.813} C_VEL
LIN {X 0,Y 429.056,Z 380.543,A -85,B 0,C 180,E1 -9637.078,E2 -9637.078} C_VEL
LIN {X 0,Y 426.571,Z 380.851,A -85,B 0,C 180,E1 -9638.099,E2 -9638.099} C_VEL
LIN {X 0,Y 425.49,Z 380.987,A -85,B 0,C 180,E1 -9638.889,E2 -9638.889} C_VEL
LIN {X 0,Y 425.399,Z 380.996,A -85,B 0,C 180,E1 -9639.156,E2 -9639.156} C_VEL
LIN {X 0,Y 425.389,Z 380.999,A -85,B 0,C 180,E1 -9642.903,E2 -9642.903} C_VEL
LIN {X 0,Y 425.357,Z 381.003,A -85,B 0,C 180,E1 -9646.605,E2 -9646.605} C_VEL
LIN {X 0,Y 425.324,Z 381.006,A -85,B 0,C 180,E1 -9649.636,E2 -9649.636} C_VEL
LIN {X 0,Y 425.302,Z 381.009,A -85,B 0,C 180,E1 -9653.365,E2 -9653.365} C_VEL
LIN {X 0,Y 425.343,Z 381.005,A -85,B 0,C 180,E1 -9656.844,E2 -9656.844} C_VEL
LIN {X 0,Y 425.313,Z 380.994,A -85,B 0,C 180,E1 -9659.717,E2 -9659.717} C_VEL
LIN {X 0,Y 425.276,Z 381.003,A -85,B 0,C 180,E1 -9663.048,E2 -9663.048} C_VEL
LIN {X 0,Y 425.278,Z 380.999,A -85,B 0,C 180,E1 -9665.929,E2 -9665.929} C_VEL
LIN {X 0,Y 425.306,Z 381.003,A -85,B 0,C 180,E1 -9669.046,E2 -9669.046} C_VEL
LIN {X 0,Y 425.308,Z 380.975,A -85,B 0,C 180,E1 -9671.962,E2 -9671.962} C_VEL
LIN {X 0,Y 425.282,Z 381.007,A -85,B 0,C 180,E1 -9675.282,E2 -9675.282} C_VEL
LIN {X 0,Y 425.296,Z 381.001,A -85,B 0,C 180,E1 -9678.625,E2 -9678.625} C_VEL
LIN {X 0,Y 425.312,Z 381.006,A -85,B 0,C 180,E1 -9681.104,E2 -9681.104} C_VEL
LIN {X 0,Y 425.293,Z 380.999,A -85,B 0,C 180,E1 -9684.664,E2 -9684.664} C_VEL
LIN {X 0,Y 425.26,Z 381.01,A -85,B 0,C 180,E1 -9688.073,E2 -9688.073} C_VEL
LIN {X 0,Y 425.331,Z 380.992,A -85,B 0,C 180,E1 -9691.369,E2 -9691.369} C_VEL
LIN {X 0,Y 425.289,Z 381.004,A -85,B 0,C 180,E1 -9694.555,E2 -9694.555} C_VEL
LIN {X 0,Y 425.281,Z 381.006,A -85,B 0,C 180,E1 -9697.662,E2 -9697.662} C_VEL
LIN {X 0,Y 425.355,Z 380.983,A -85,B 0,C 180,E1 -9700.704,E2 -9700.704} C_VEL
LIN {X 0,Y 425.381,Z 380.991,A -85,B 0,C 180,E1 -9703.689,E2 -9703.689} C_VEL
LIN {X 0,Y 425.423,Z 380.984,A -85,B 0,C 180,E1 -9707.599,E2 -9707.599} C_VEL
LIN {X 0,Y 425.436,Z 380.976,A -85,B 0,C 180,E1 -9711.45,E2 -9711.45} C_VEL
LIN {X 0,Y 425.548,Z 380.978,A -85,B 0,C 180,E1 -9714.314,E2 -9714.314} C_VEL
LIN {X 0,Y 425.57,Z 380.962,A -85,B 0,C 180,E1 -9718.108,E2 -9718.108} C_VEL
LIN {X 0,Y 425.697,Z 380.935,A -85,B 0,C 180,E1 -9720.001,E2 -9720.001} C_VEL
LIN {X 0,Y 425.552,Z 380.973,A -85,B 0,C 180,E1 -9722.84,E2 -9722.84} C_VEL
LIN {X 0,Y 425.525,Z 380.972,A -85,B 0,C 180,E1 -9726.639,E2 -9726.639} C_VEL
LIN {X 0,Y 425.396,Z 380.97,A -85,B 0,C 180,E1 -9729.51,E2 -9729.51} C_VEL
LIN {X 0,Y 425.388,Z 380.992,A -85,B 0,C 180,E1 -9732.904,E2 -9732.904} C_VEL
LIN {X 0,Y 425.365,Z 380.987,A -85,B 0,C 180,E1 -9736.61,E2 -9736.61} C_VEL
LIN {X 0,Y 425.324,Z 380.987,A -85,B 0,C 180,E1 -9739.636,E2 -9739.636} C_VEL
LIN {X 0,Y 425.303,Z 381.003,A -85,B 0,C 180,E1 -9743.366,E2 -9743.366} C_VEL
LIN {X 0,Y 425.345,Z 380.986,A -85,B 0,C 180,E1 -9746.845,E2 -9746.845} C_VEL
LIN {X 0,Y 425.315,Z 381.003,A -85,B 0,C 180,E1 -9749.718,E2 -9749.718} C_VEL
LIN {X 0,Y 425.281,Z 380.999,A -85,B 0,C 180,E1 -9753.049,E2 -9753.049} C_VEL
LIN {X 0,Y 425.282,Z 381.007,A -85,B 0,C 180,E1 -9755.93,E2 -9755.93} C_VEL
LIN {X 0,Y 425.308,Z 380.999,A -85,B 0,C 180,E1 -9759.046,E2 -9759.046} C_VEL
LIN {X 0,Y 425.33,Z 381.001,A -85,B 0,C 180,E1 -9762.647,E2 -9762.647} C_VEL
LIN {X 0,Y 425.293,Z 381.005,A -85,B 0,C 180,E1 -9765.283,E2 -9765.283} C_VEL
LIN {X 0,Y 425.273,Z 380.995,A -85,B 0,C 180,E1 -9768.622,E2 -9768.622} C_VEL
LIN {X 0,Y 425.313,Z 381.002,A -85,B 0,C 180,E1 -9771.104,E2 -9771.104} C_VEL
LIN {X 0,Y 425.301,Z 381.002,A -85,B 0,C 180,E1 -9774.665,E2 -9774.665} C_VEL
LIN {X 0,Y 425.273,Z 381.009,A -85,B 0,C 180,E1 -9778.075,E2 -9778.075} C_VEL
LIN {X 0,Y 425.36,Z 381.14,A -85,B 0,C 180,E1 -9781.05,E2 -9781.05} C_VEL
LIN {X 0,Y 427.128,Z 390.321,A -85,B 0,C 180,E1 -9783.625,E2 -9783.625} C_VEL
LIN {X 0,Y 427.663,Z 395.42,A -85,B 0,C 180,E1 -9784.966,E2 -9784.966} C_VEL
LIN {X 0,Y 426.82,Z 408.885,A -85,B 0,C 180,E1 -9788.255,E2 -9788.255} C_VEL
LIN {X 0,Y 426.074,Z 420.938,A -85,B 0,C 180,E1 -9791.207,E2 -9791.207} C_VEL
LIN {X 0,Y 426.64,Z 424.373,A -85,B 0,C 180,E1 -9791.345,E2 -9791.345} C_VEL
LIN {X 0,Y 430.494,Z 446.691,A -85,B 0,C 180,E1 -9791.9,E2 -9791.9} C_VEL
LIN {X 0,Y 429.684,Z 525.884,A -85,B 0,C 180,E1 -9793.246,E2 -9793.246} C_VEL
LIN {X 0,Y 429.392,Z 535.797,A -85,B 0,C 180,E1 -9793.509,E2 -9793.509} C_VEL
LIN {X 0,Y 428.935,Z 545.782,A -85,B 0,C 180,E1 -9793.888,E2 -9793.888} C_VEL
LIN {X 0,Y 428.418,Z 556.14,A -85,B 0,C 180,E1 -9794.418,E2 -9794.418} C_VEL
LIN {X 0,Y 427.865,Z 565.286,A -85,B 0,C 180,E1 -9795.007,E2 -9795.007} C_VEL
LIN {X 0,Y 427.323,Z 574.29,A -85,B 0,C 180,E1 -9795.718,E2 -9795.718} C_VEL
LIN {X 0,Y 426.794,Z 582.236,A -85,B 0,C 180,E1 -9796.464,E2 -9796.464} C_VEL
LIN {X 0,Y 426.294,Z 590.443,A -85,B 0,C 180,E1 -9797.383,E2 -9797.383} C_VEL
LIN {X 0,Y 425.643,Z 599.24,A -85,B 0,C 180,E1 -9798.572,E2 -9798.572} C_VEL
LIN {X 0,Y 425.2,Z 605.23,A -85,B 0,C 180,E1 -9799.525,E2 -9799.525} C_VEL
LIN {X 0,Y 424.817,Z 611.542,A -85,B 0,C 180,E1 -9800.718,E2 -9800.718} C_VEL
LIN {X 0,Y 424.533,Z 616.816,A -85,B 0,C 180,E1 -9801.911,E2 -9801.911} C_VEL
LIN {X 0,Y 424.302,Z 621.908,A -85,B 0,C 180,E1 -9803.342,E2 -9803.342} C_VEL
LIN {X 0,Y 424.21,Z 625.871,A -85,B 0,C 180,E1 -9804.772,E2 -9804.772} C_VEL
LIN {X 0,Y 424.099,Z 628.801,A -85,B 0,C 180,E1 -9806.2,E2 -9806.2} C_VEL
LIN {X 0,Y 424.131,Z 630.301,A -85,B 0,C 180,E1 -9807.151,E2 -9807.151} C_VEL
LIN {X 0,Y 424.089,Z 631.82,A -85,B 0,C 180,E1 -9809.051,E2 -9809.051} C_VEL
LIN {X 0,Y 424.084,Z 632.098,A -85,B 0,C 180,E1 -9810,E2 -9810} C_VEL
LIN {X 0,Y 424.129,Z 631.226,A -85,B 0,C 180,E1 -9811.899,E2 -9811.899} C_VEL
LIN {X 0,Y 424.132,Z 630.3,A -85,B 0,C 180,E1 -9812.85,E2 -9812.85} C_VEL
LIN {X 0,Y 424.201,Z 626.958,A -85,B 0,C 180,E1 -9814.752,E2 -9814.752} C_VEL
LIN {X 0,Y 424.195,Z 624.745,A -85,B 0,C 180,E1 -9815.705,E2 -9815.705} C_VEL
LIN {X 0,Y 424.359,Z 620.392,A -85,B 0,C 180,E1 -9817.135,E2 -9817.135} C_VEL
LIN {X 0,Y 424.642,Z 614.817,A -85,B 0,C 180,E1 -9818.566,E2 -9818.566} C_VEL
LIN {X 0,Y 424.954,Z 609.163,A -85,B 0,C 180,E1 -9819.76,E2 -9819.76} C_VEL
LIN {X 0,Y 425.391,Z 602.357,A -85,B 0,C 180,E1 -9820.953,E2 -9820.953} C_VEL
LIN {X 0,Y 426.02,Z 594.14,A -85,B 0,C 180,E1 -9822.142,E2 -9822.142} C_VEL
LIN {X 0,Y 426.534,Z 586.31,A -85,B 0,C 180,E1 -9823.095,E2 -9823.095} C_VEL
LIN {X 0,Y 427.075,Z 578.231,A -85,B 0,C 180,E1 -9823.926,E2 -9823.926} C_VEL
LIN {X 0,Y 427.69,Z 568.459,A -85,B 0,C 180,E1 -9824.756,E2 -9824.756} C_VEL
LIN {X 0,Y 428.177,Z 560.067,A -85,B 0,C 180,E1 -9825.348,E2 -9825.348} C_VEL
LIN {X 0,Y 428.794,Z 549.56,A -85,B 0,C 180,E1 -9825.934,E2 -9825.934} C_VEL
LIN {X 0,Y 429.213,Z 539.224,A -85,B 0,C 180,E1 -9826.376,E2 -9826.376} C_VEL
LIN {X 0,Y 429.665,Z 528.503,A -85,B 0,C 180,E1 -9826.695,E2 -9826.695} C_VEL
LIN {X 0,Y 429.958,Z 505.724,A -85,B 0,C 180,E1 -9827.111,E2 -9827.111} C_VEL
LIN {X 0,Y 430.399,Z 445.696,A -85,B 0,C 180,E1 -9828.122,E2 -9828.122} C_VEL
LIN {X 0,Y 426.084,Z 421.205,A -85,B 0,C 180,E1 -9828.762,E2 -9828.762} C_VEL
LIN {X 0,Y 426.127,Z 419.896,A -85,B 0,C 180,E1 -9829.01,E2 -9829.01} C_VEL
LIN {X 0,Y 427.054,Z 405.759,A -85,B 0,C 180,E1 -9832.553,E2 -9832.553} C_VEL
LIN {X 0,Y 427.743,Z 394.393,A -85,B 0,C 180,E1 -9835.354,E2 -9835.354} C_VEL
LIN {X 0,Y 426.383,Z 386.337,A -85,B 0,C 180,E1 -9837.485,E2 -9837.485} C_VEL
LIN {X 0,Y 425.356,Z 381.105,A -85,B 0,C 180,E1 -9838.983,E2 -9838.983} C_VEL
LIN {X 0,Y 425.288,Z 381.003,A -85,B 0,C 180,E1 -9842.563,E2 -9842.563} C_VEL
LIN {X 0,Y 425.303,Z 381.002,A -85,B 0,C 180,E1 -9845.335,E2 -9845.335} C_VEL
LIN {X 0,Y 425.315,Z 381.002,A -85,B 0,C 180,E1 -9848.897,E2 -9848.897} C_VEL
LIN {X 0,Y 425.291,Z 380.998,A -85,B 0,C 180,E1 -9851.958,E2 -9851.958} C_VEL
LIN {X 0,Y 425.315,Z 381.002,A -85,B 0,C 180,E1 -9855.279,E2 -9855.279} C_VEL
LIN {X 0,Y 425.311,Z 381.002,A -85,B 0,C 180,E1 -9858.625,E2 -9858.625} C_VEL
LIN {X 0,Y 425.323,Z 380.997,A -85,B 0,C 180,E1 -9861.103,E2 -9861.103} C_VEL
LIN {X 0,Y 425.301,Z 380.999,A -85,B 0,C 180,E1 -9864.664,E2 -9864.664} C_VEL
LIN {X 0,Y 425.273,Z 381.011,A -85,B 0,C 180,E1 -9868.073,E2 -9868.073} C_VEL
LIN {X 0,Y 425.338,Z 381,A -85,B 0,C 180,E1 -9871.368,E2 -9871.368} C_VEL
LIN {X 0,Y 425.295,Z 380.998,A -85,B 0,C 180,E1 -9874.554,E2 -9874.554} C_VEL
LIN {X 0,Y 425.287,Z 381.01,A -85,B 0,C 180,E1 -9877.661,E2 -9877.661} C_VEL
LIN {X 0,Y 425.361,Z 380.981,A -85,B 0,C 180,E1 -9880.703,E2 -9880.703} C_VEL
LIN {X 0,Y 425.398,Z 380.987,A -85,B 0,C 180,E1 -9883.688,E2 -9883.688} C_VEL
LIN {X 0,Y 425.411,Z 380.991,A -85,B 0,C 180,E1 -9887.598,E2 -9887.598} C_VEL
LIN {X 0,Y 425.441,Z 380.967,A -85,B 0,C 180,E1 -9891.449,E2 -9891.449} C_VEL
LIN {X 0,Y 425.552,Z 380.973,A -85,B 0,C 180,E1 -9894.313,E2 -9894.313} C_VEL
LIN {X 0,Y 425.573,Z 380.963,A -85,B 0,C 180,E1 -9898.107,E2 -9898.107} C_VEL
LIN {X 0,Y 425.699,Z 380.935,A -85,B 0,C 180,E1 -9899.999,E2 -9899.999} C_VEL
LIN {X 0,Y 425.555,Z 380.966,A -85,B 0,C 180,E1 -9902.839,E2 -9902.839} C_VEL
LIN {X 0,Y 425.528,Z 380.974,A -85,B 0,C 180,E1 -9906.646,E2 -9906.646} C_VEL
LIN {X 0,Y 425.4,Z 380.976,A -85,B 0,C 180,E1 -9909.509,E2 -9909.509} C_VEL
LIN {X 0,Y 425.401,Z 380.988,A -85,B 0,C 180,E1 -9912.91,E2 -9912.91} C_VEL
LIN {X 0,Y 425.358,Z 380.994,A -85,B 0,C 180,E1 -9916.605,E2 -9916.605} C_VEL
LIN {X 0,Y 425.325,Z 380.988,A -85,B 0,C 180,E1 -9919.635,E2 -9919.635} C_VEL
LIN {X 0,Y 425.304,Z 381.009,A -85,B 0,C 180,E1 -9923.365,E2 -9923.365} C_VEL
LIN {X 0,Y 425.345,Z 380.99,A -85,B 0,C 180,E1 -9926.844,E2 -9926.844} C_VEL
LIN {X 0,Y 425.287,Z 381.01,A -85,B 0,C 180,E1 -9929.719,E2 -9929.719} C_VEL
LIN {X 0,Y 425.278,Z 381.009,A -85,B 0,C 180,E1 -9933.048,E2 -9933.048} C_VEL
LIN {X 0,Y 425.28,Z 381.007,A -85,B 0,C 180,E1 -9935.929,E2 -9935.929} C_VEL
LIN {X 0,Y 425.297,Z 381.009,A -85,B 0,C 180,E1 -9939.044,E2 -9939.044} C_VEL
LIN {X 0,Y 425.274,Z 381.007,A -85,B 0,C 180,E1 -9942.652,E2 -9942.652} C_VEL
LIN {X 0,Y 425.257,Z 380.997,A -85,B 0,C 180,E1 -9946.044,E2 -9946.044} C_VEL
LIN {X 0,Y 425.3,Z 380.978,A -85,B 0,C 180,E1 -9948.625,E2 -9948.625} C_VEL
LIN {X 0,Y 425.32,Z 381.003,A -85,B 0,C 180,E1 -9951.104,E2 -9951.104} C_VEL
LIN {X 0,Y 425.297,Z 380.994,A -85,B 0,C 180,E1 -9954.664,E2 -9954.664} C_VEL
LIN {X 0,Y 425.263,Z 381.011,A -85,B 0,C 180,E1 -9958.073,E2 -9958.073} C_VEL
LIN {X 0,Y 425.334,Z 380.994,A -85,B 0,C 180,E1 -9961.368,E2 -9961.368} C_VEL
LIN {X 0,Y 425.292,Z 381.009,A -85,B 0,C 180,E1 -9964.554,E2 -9964.554} C_VEL
LIN {X 0,Y 425.284,Z 381.012,A -85,B 0,C 180,E1 -9967.661,E2 -9967.661} C_VEL
LIN {X 0,Y 425.359,Z 381.002,A -85,B 0,C 180,E1 -9970.704,E2 -9970.704} C_VEL
LIN {X 0,Y 425.385,Z 380.999,A -85,B 0,C 180,E1 -9973.688,E2 -9973.688} C_VEL
LIN {X 0,Y 425.408,Z 380.996,A -85,B 0,C 180,E1 -9977.598,E2 -9977.598} C_VEL
LIN {X 0,Y 425.439,Z 380.993,A -85,B 0,C 180,E1 -9981.45,E2 -9981.45} C_VEL
LIN {X 0,Y 425.552,Z 380.978,A -85,B 0,C 180,E1 -9984.313,E2 -9984.313} C_VEL
LIN {X 0,Y 425.572,Z 380.975,A -85,B 0,C 180,E1 -9988.107,E2 -9988.107} C_VEL
LIN {X 0,Y 425.7,Z 380.96,A -85,B 0,C 180,E1 -9990,E2 -9990} C_VEL
LIN {X 0,Y 425.553,Z 380.978,A -85,B 0,C 180,E1 -9992.84,E2 -9992.84} C_VEL
LIN {X 0,Y 425.528,Z 380.982,A -85,B 0,C 180,E1 -9996.639,E2 -9996.639} C_VEL
LIN {X 0,Y 425.399,Z 380.996,A -85,B 0,C 180,E1 -9999.156,E2 -9999.156} C_VEL
LIN {X 0,Y 424.727,Z 381.081,A -85,B 0,C 180,E1 -9999.946,E2 -9999.946} C_VEL
LIN {X 0,Y 421.878,Z 381.437,A -85,B 0,C 180,E1 -10001.23,E2 -10001.23} C_VEL
LIN {X 0,Y 419.462,Z 381.738,A -85,B 0,C 180,E1 -10002.266,E2 -10002.266} C_VEL
LIN {X 0,Y 418.411,Z 381.869,A -85,B 0,C 180,E1 -10003.067,E2 -10003.067} C_VEL
LIN {X 0,Y 418.318,Z 381.879,A -85,B 0,C 180,E1 -10003.338,E2 -10003.338} C_VEL
LIN {X 0,Y 418.308,Z 381.881,A -85,B 0,C 180,E1 -10006.735,E2 -10006.735} C_VEL
LIN {X 0,Y 418.266,Z 381.885,A -85,B 0,C 180,E1 -10009.79,E2 -10009.79} C_VEL
LIN {X 0,Y 418.233,Z 381.891,A -85,B 0,C 180,E1 -10012.736,E2 -10012.736} C_VEL
LIN {X 0,Y 418.266,Z 381.884,A -85,B 0,C 180,E1 -10015.904,E2 -10015.904} C_VEL
LIN {X 0,Y 418.269,Z 381.87,A -85,B 0,C 180,E1 -10019.161,E2 -10019.161} C_VEL
LIN {X 0,Y 418.252,Z 381.88,A -85,B 0,C 180,E1 -10022.844,E2 -10022.844} C_VEL
LIN {X 0,Y 418.243,Z 381.877,A -85,B 0,C 180,E1 -10026.239,E2 -10026.239} C_VEL
LIN {X 0,Y 418.259,Z 381.877,A -85,B 0,C 180,E1 -10029.68,E2 -10029.68} C_VEL
LIN {X 0,Y 418.238,Z 381.855,A -85,B 0,C 180,E1 -10032.323,E2 -10032.323} C_VEL
LIN {X 0,Y 418.232,Z 381.887,A -85,B 0,C 180,E1 -10035.109,E2 -10035.109} C_VEL
LIN {X 0,Y 418.251,Z 381.882,A -85,B 0,C 180,E1 -10037.769,E2 -10037.769} C_VEL
LIN {X 0,Y 418.257,Z 381.881,A -85,B 0,C 180,E1 -10040.617,E2 -10040.617} C_VEL
LIN {X 0,Y 418.239,Z 381.883,A -85,B 0,C 180,E1 -10043.976,E2 -10043.976} C_VEL
LIN {X 0,Y 418.251,Z 381.883,A -85,B 0,C 180,E1 -10047.156,E2 -10047.156} C_VEL
LIN {X 0,Y 418.267,Z 381.876,A -85,B 0,C 180,E1 -10050.839,E2 -10050.839} C_VEL
LIN {X 0,Y 418.264,Z 381.873,A -85,B 0,C 180,E1 -10054.096,E2 -10054.096} C_VEL
LIN {X 0,Y 418.231,Z 381.884,A -85,B 0,C 180,E1 -10057.264,E2 -10057.264} C_VEL
LIN {X 0,Y 418.276,Z 381.865,A -85,B 0,C 180,E1 -10060.364,E2 -10060.364} C_VEL
LIN {X 0,Y 418.31,Z 381.872,A -85,B 0,C 180,E1 -10063.405,E2 -10063.405} C_VEL
LIN {X 0,Y 418.348,Z 381.867,A -85,B 0,C 180,E1 -10066.994,E2 -10066.994} C_VEL
LIN {X 0,Y 418.337,Z 381.854,A -85,B 0,C 180,E1 -10070.329,E2 -10070.329} C_VEL
LIN {X 0,Y 418.487,Z 381.851,A -85,B 0,C 180,E1 -10073.249,E2 -10073.249} C_VEL
LIN {X 0,Y 418.336,Z 381.872,A -85,B 0,C 180,E1 -10075.182,E2 -10075.182} C_VEL
LIN {X 0,Y 418.539,Z 381.837,A -85,B 0,C 180,E1 -10078.076,E2 -10078.076} C_VEL
LIN {X 0,Y 418.666,Z 381.81,A -85,B 0,C 180,E1 -10080.001,E2 -10080.001} C_VEL
LIN {X 0,Y 418.506,Z 381.851,A -85,B 0,C 180,E1 -10082.888,E2 -10082.888} C_VEL
LIN {X 0,Y 418.488,Z 381.847,A -85,B 0,C 180,E1 -10086.752,E2 -10086.752} C_VEL
LIN {X 0,Y 418.395,Z 381.844,A -85,B 0,C 180,E1 -10088.696,E2 -10088.696} C_VEL
LIN {X 0,Y 418.31,Z 381.866,A -85,B 0,C 180,E1 -10091.632,E2 -10091.632} C_VEL
LIN {X 0,Y 418.302,Z 381.876,A -85,B 0,C 180,E1 -10094.598,E2 -10094.598} C_VEL
LIN {X 0,Y 418.284,Z 381.867,A -85,B 0,C 180,E1 -10097.604,E2 -10097.604} C_VEL
LIN {X 0,Y 418.246,Z 381.881,A -85,B 0,C 180,E1 -10100.664,E2 -10100.664} C_VEL
LIN {X 0,Y 418.284,Z 381.88,A -85,B 0,C 180,E1 -10103.782,E2 -10103.782} C_VEL
LIN {X 0,Y 418.306,Z 381.861,A -85,B 0,C 180,E1 -10107.071,E2 -10107.071} C_VEL
LIN {X 0,Y 418.259,Z 381.887,A -85,B 0,C 180,E1 -10110.271,E2 -10110.271} C_VEL
LIN {X 0,Y 418.247,Z 381.875,A -85,B 0,C 180,E1 -10113.678,E2 -10113.678} C_VEL
LIN {X 0,Y 418.244,Z 381.884,A -85,B 0,C 180,E1 -10117.224,E2 -10117.224} C_VEL
LIN {X 0,Y 418.263,Z 381.878,A -85,B 0,C 180,E1 -10119.681,E2 -10119.681} C_VEL
LIN {X 0,Y 418.284,Z 381.882,A -85,B 0,C 180,E1 -10122.33,E2 -10122.33} C_VEL
LIN {X 0,Y 418.25,Z 381.882,A -85,B 0,C 180,E1 -10125.112,E2 -10125.112} C_VEL
LIN {X 0,Y 418.239,Z 381.882,A -85,B 0,C 180,E1 -10127.768,E2 -10127.768} C_VEL
LIN {X 0,Y 418.256,Z 381.881,A -85,B 0,C 180,E1 -10130.619,E2 -10130.619} C_VEL
LIN {X 0,Y 418.246,Z 381.877,A -85,B 0,C 180,E1 -10133.977,E2 -10133.977} C_VEL
LIN {X 0,Y 418.261,Z 381.878,A -85,B 0,C 180,E1 -10137.156,E2 -10137.156} C_VEL
LIN {X 0,Y 418.309,Z 382.06,A -85,B 0,C 180,E1 -10140.808,E2 -10140.808} C_VEL
LIN {X 0,Y 420.251,Z 392.114,A -85,B 0,C 180,E1 -10143.694,E2 -10143.694} C_VEL
LIN {X 0,Y 420.718,Z 396.65,A -85,B 0,C 180,E1 -10144.882,E2 -10144.882} C_VEL
LIN {X 0,Y 419.756,Z 410.782,A -85,B 0,C 180,E1 -10148.387,E2 -10148.387} C_VEL
LIN {X 0,Y 419.113,Z 420.741,A -85,B 0,C 180,E1 -10150.883,E2 -10150.883} C_VEL
LIN {X 0,Y 419.658,Z 424.117,A -85,B 0,C 180,E1 -10151.022,E2 -10151.022} C_VEL
LIN {X 0,Y 423.71,Z 447.294,A -85,B 0,C 180,E1 -10151.614,E2 -10151.614} C_VEL
LIN {X 0,Y 422.898,Z 525.689,A -85,B 0,C 180,E1 -10152.969,E2 -10152.969} C_VEL
LIN {X 0,Y 422.582,Z 535.602,A -85,B 0,C 180,E1 -10153.236,E2 -10153.236} C_VEL
LIN {X 0,Y 422.129,Z 545.588,A -85,B 0,C 180,E1 -10153.621,E2 -10153.621} C_VEL
LIN {X 0,Y 421.593,Z 555.945,A -85,B 0,C 180,E1 -10154.159,E2 -10154.159} C_VEL
LIN {X 0,Y 421.002,Z 565.09,A -85,B 0,C 180,E1 -10154.757,E2 -10154.757} C_VEL
LIN {X 0,Y 420.419,Z 574.094,A -85,B 0,C 180,E1 -10155.479,E2 -10155.479} C_VEL
LIN {X 0,Y 419.821,Z 582.8,A -85,B 0,C 180,E1 -10156.32,E2 -10156.32} C_VEL
LIN {X 0,Y 419.341,Z 590.248,A -85,B 0,C 180,E1 -10157.17,E2 -10157.17} C_VEL
LIN {X 0,Y 418.645,Z 599.044,A -85,B 0,C 180,E1 -10158.379,E2 -10158.379} C_VEL
LIN {X 0,Y 418.175,Z 605.034,A -85,B 0,C 180,E1 -10159.347,E2 -10159.347} C_VEL
LIN {X 0,Y 417.782,Z 611.346,A -85,B 0,C 180,E1 -10160.56,E2 -10160.56} C_VEL
LIN {X 0,Y 417.471,Z 616.62,A -85,B 0,C 180,E1 -10161.773,E2 -10161.773} C_VEL
LIN {X 0,Y 417.235,Z 621.713,A -85,B 0,C 180,E1 -10163.229,E2 -10163.229} C_VEL
LIN {X 0,Y 417.125,Z 625.676,A -85,B 0,C 180,E1 -10164.683,E2 -10164.683} C_VEL
LIN {X 0,Y 417.014,Z 628.606,A -85,B 0,C 180,E1 -10166.135,E2 -10166.135} C_VEL
LIN {X 0,Y 417.028,Z 630.105,A -85,B 0,C 180,E1 -10167.102,E2 -10167.102} C_VEL
LIN {X 0,Y 417.011,Z 631.625,A -85,B 0,C 180,E1 -10169.035,E2 -10169.035} C_VEL
LIN {X 0,Y 417.004,Z 631.903,A -85,B 0,C 180,E1 -10170,E2 -10170} C_VEL
LIN {X 0,Y 417.057,Z 631.032,A -85,B 0,C 180,E1 -10171.932,E2 -10171.932} C_VEL
LIN {X 0,Y 417.028,Z 630.105,A -85,B 0,C 180,E1 -10172.898,E2 -10172.898} C_VEL
LIN {X 0,Y 417.109,Z 626.763,A -85,B 0,C 180,E1 -10174.833,E2 -10174.833} C_VEL
LIN {X 0,Y 417.144,Z 623.212,A -85,B 0,C 180,E1 -10176.262,E2 -10176.262} C_VEL
LIN {X 0,Y 417.375,Z 618.408,A -85,B 0,C 180,E1 -10177.742,E2 -10177.742} C_VEL
LIN {X 0,Y 417.693,Z 612.436,A -85,B 0,C 180,E1 -10179.198,E2 -10179.198} C_VEL
LIN {X 0,Y 418.105,Z 606.343,A -85,B 0,C 180,E1 -10180.411,E2 -10180.411} C_VEL
LIN {X 0,Y 418.502,Z 600.6,A -85,B 0,C 180,E1 -10181.38,E2 -10181.38} C_VEL
LIN {X 0,Y 419.059,Z 593.945,A -85,B 0,C 180,E1 -10182.347,E2 -10182.347} C_VEL
LIN {X 0,Y 419.603,Z 586.115,A -85,B 0,C 180,E1 -10183.315,E2 -10183.315} C_VEL
LIN {X 0,Y 420.2,Z 577.405,A -85,B 0,C 180,E1 -10184.217,E2 -10184.217} C_VEL
LIN {X 0,Y 420.807,Z 568.264,A -85,B 0,C 180,E1 -10185.003,E2 -10185.003} C_VEL
LIN {X 0,Y 421.319,Z 559.871,A -85,B 0,C 180,E1 -10185.604,E2 -10185.604} C_VEL
LIN {X 0,Y 421.96,Z 549.364,A -85,B 0,C 180,E1 -10186.2,E2 -10186.2} C_VEL
LIN {X 0,Y 422.404,Z 539.029,A -85,B 0,C 180,E1 -10186.648,E2 -10186.648} C_VEL
LIN {X 0,Y 422.885,Z 528.309,A -85,B 0,C 180,E1 -10186.97,E2 -10186.97} C_VEL
LIN {X 0,Y 423.184,Z 505.529,A -85,B 0,C 180,E1 -10187.394,E2 -10187.394} C_VEL
LIN {X 0,Y 423.649,Z 446.445,A -85,B 0,C 180,E1 -10188.404,E2 -10188.404} C_VEL
LIN {X 0,Y 419.132,Z 421.01,A -85,B 0,C 180,E1 -10189.085,E2 -10189.085} C_VEL
LIN {X 0,Y 419.154,Z 419.701,A -85,B 0,C 180,E1 -10189.338,E2 -10189.338} C_VEL
LIN {X 0,Y 420.067,Z 406.851,A -85,B 0,C 180,E1 -10192.632,E2 -10192.632} C_VEL
LIN {X 0,Y 420.781,Z 396.87,A -85,B 0,C 180,E1 -10195.125,E2 -10195.125} C_VEL
LIN {X 0,Y 420.33,Z 392.4,A -85,B 0,C 180,E1 -10196.301,E2 -10196.301} C_VEL
LIN {X 0,Y 418.305,Z 381.99,A -85,B 0,C 180,E1 -10199.228,E2 -10199.228} C_VEL
LIN {X 0,Y 418.263,Z 381.878,A -85,B 0,C 180,E1 -10202.844,E2 -10202.844} C_VEL
LIN {X 0,Y 418.251,Z 381.877,A -85,B 0,C 180,E1 -10206.238,E2 -10206.238} C_VEL
LIN {X 0,Y 418.254,Z 381.875,A -85,B 0,C 180,E1 -10209.681,E2 -10209.681} C_VEL
LIN {X 0,Y 418.231,Z 381.884,A -85,B 0,C 180,E1 -10212.321,E2 -10212.321} C_VEL
LIN {X 0,Y 418.26,Z 381.88,A -85,B 0,C 180,E1 -10215.111,E2 -10215.111} C_VEL
LIN {X 0,Y 418.294,Z 381.882,A -85,B 0,C 180,E1 -10217.773,E2 -10217.773} C_VEL
LIN {X 0,Y 418.266,Z 381.879,A -85,B 0,C 180,E1 -10221.559,E2 -10221.559} C_VEL
LIN {X 0,Y 418.26,Z 381.876,A -85,B 0,C 180,E1 -10225.159,E2 -10225.159} C_VEL
LIN {X 0,Y 418.25,Z 381.877,A -85,B 0,C 180,E1 -10227.472,E2 -10227.472} C_VEL
LIN {X 0,Y 418.277,Z 381.877,A -85,B 0,C 180,E1 -10230.893,E2 -10230.893} C_VEL
LIN {X 0,Y 418.271,Z 381.871,A -85,B 0,C 180,E1 -10234.095,E2 -10234.095} C_VEL
LIN {X 0,Y 418.238,Z 381.884,A -85,B 0,C 180,E1 -10237.263,E2 -10237.263} C_VEL
LIN {X 0,Y 418.282,Z 381.864,A -85,B 0,C 180,E1 -10240.364,E2 -10240.364} C_VEL
LIN {X 0,Y 418.325,Z 381.864,A -85,B 0,C 180,E1 -10243.404,E2 -10243.404} C_VEL
LIN {X 0,Y 418.345,Z 381.869,A -85,B 0,C 180,E1 -10246.999,E2 -10246.999} C_VEL
LIN {X 0,Y 418.34,Z 381.846,A -85,B 0,C 180,E1 -10250.328,E2 -10250.328} C_VEL
LIN {X 0,Y 418.512,Z 381.843,A -85,B 0,C 180,E1 -10252.279,E2 -10252.279} C_VEL
LIN {X 0,Y 418.511,Z 381.851,A -85,B 0,C 180,E1 -10254.217,E2 -10254.217} C_VEL
LIN {X 0,Y 418.543,Z 381.838,A -85,B 0,C 180,E1 -10258.075,E2 -10258.075} C_VEL
LIN {X 0,Y 418.668,Z 381.81,A -85,B 0,C 180,E1 -10259.999,E2 -10259.999} C_VEL
LIN {X 0,Y 418.509,Z 381.843,A -85,B 0,C 180,E1 -10262.887,E2 -10262.887} C_VEL
LIN {X 0,Y 418.491,Z 381.851,A -85,B 0,C 180,E1 -10266.75,E2 -10266.75} C_VEL
LIN {X 0,Y 418.341,Z 381.853,A -85,B 0,C 180,E1 -10269.671,E2 -10269.671} C_VEL
LIN {X 0,Y 418.352,Z 381.866,A -85,B 0,C 180,E1 -10273.006,E2 -10273.006} C_VEL
LIN {X 0,Y 418.31,Z 381.872,A -85,B 0,C 180,E1 -10276.735,E2 -10276.735} C_VEL
LIN {X 0,Y 418.267,Z 381.868,A -85,B 0,C 180,E1 -10279.79,E2 -10279.79} C_VEL
LIN {X 0,Y 418.235,Z 381.884,A -85,B 0,C 180,E1 -10282.736,E2 -10282.736} C_VEL
LIN {X 0,Y 418.268,Z 381.873,A -85,B 0,C 180,E1 -10285.904,E2 -10285.904} C_VEL
LIN {X 0,Y 418.261,Z 381.876,A -85,B 0,C 180,E1 -10289.162,E2 -10289.162} C_VEL
LIN {X 0,Y 418.254,Z 381.883,A -85,B 0,C 180,E1 -10292.844,E2 -10292.844} C_VEL
LIN {X 0,Y 418.244,Z 381.882,A -85,B 0,C 180,E1 -10296.238,E2 -10296.238} C_VEL
LIN {X 0,Y 418.248,Z 381.878,A -85,B 0,C 180,E1 -10299.681,E2 -10299.681} C_VEL
LIN {X 0,Y 418.228,Z 381.884,A -85,B 0,C 180,E1 -10302.321,E2 -10302.321} C_VEL
LIN {X 0,Y 418.234,Z 381.883,A -85,B 0,C 180,E1 -10305.109,E2 -10305.109} C_VEL
LIN {X 0,Y 418.252,Z 381.853,A -85,B 0,C 180,E1 -10307.769,E2 -10307.769} C_VEL
LIN {X 0,Y 418.264,Z 381.877,A -85,B 0,C 180,E1 -10310.616,E2 -10310.616} C_VEL
LIN {X 0,Y 418.242,Z 381.876,A -85,B 0,C 180,E1 -10313.976,E2 -10313.976} C_VEL
LIN {X 0,Y 418.254,Z 381.88,A -85,B 0,C 180,E1 -10317.156,E2 -10317.156} C_VEL
LIN {X 0,Y 418.271,Z 381.87,A -85,B 0,C 180,E1 -10320.839,E2 -10320.839} C_VEL
LIN {X 0,Y 418.267,Z 381.883,A -85,B 0,C 180,E1 -10324.096,E2 -10324.096} C_VEL
LIN {X 0,Y 418.235,Z 381.891,A -85,B 0,C 180,E1 -10327.264,E2 -10327.264} C_VEL
LIN {X 0,Y 418.28,Z 381.883,A -85,B 0,C 180,E1 -10330.364,E2 -10330.364} C_VEL
LIN {X 0,Y 418.314,Z 381.881,A -85,B 0,C 180,E1 -10333.404,E2 -10333.404} C_VEL
LIN {X 0,Y 418.343,Z 381.877,A -85,B 0,C 180,E1 -10336.999,E2 -10336.999} C_VEL
LIN {X 0,Y 418.338,Z 381.876,A -85,B 0,C 180,E1 -10340.328,E2 -10340.328} C_VEL
LIN {X 0,Y 418.491,Z 381.858,A -85,B 0,C 180,E1 -10343.249,E2 -10343.249} C_VEL
LIN {X 0,Y 418.338,Z 381.878,A -85,B 0,C 180,E1 -10345.181,E2 -10345.181} C_VEL
LIN {X 0,Y 418.541,Z 381.851,A -85,B 0,C 180,E1 -10348.075,E2 -10348.075} C_VEL
LIN {X 0,Y 418.669,Z 381.836,A -85,B 0,C 180,E1 -10350,E2 -10350} C_VEL
LIN {X 0,Y 418.507,Z 381.856,A -85,B 0,C 180,E1 -10352.887,E2 -10352.887} C_VEL
LIN {X 0,Y 418.491,Z 381.858,A -85,B 0,C 180,E1 -10356.751,E2 -10356.751} C_VEL
LIN {X 0,Y 418.337,Z 381.876,A -85,B 0,C 180,E1 -10359.671,E2 -10359.671} C_VEL
LIN {X 0,Y 418.318,Z 381.879,A -85,B 0,C 180,E1 -10363.338,E2 -10363.338} C_VEL
LIN {X 0,Y 417.624,Z 381.966,A -85,B 0,C 180,E1 -10364.141,E2 -10364.141} C_VEL
LIN {X 0,Y 414.746,Z 382.325,A -85,B 0,C 180,E1 -10365.447,E2 -10365.447} C_VEL
LIN {X 0,Y 412.333,Z 382.626,A -85,B 0,C 180,E1 -10366.501,E2 -10366.501} C_VEL
LIN {X 0,Y 411.312,Z 382.752,A -85,B 0,C 180,E1 -10367.316,E2 -10367.316} C_VEL
LIN {X 0,Y 411.235,Z 382.76,A -85,B 0,C 180,E1 -10367.592,E2 -10367.592} C_VEL
LIN {X 0,Y 411.192,Z 382.768,A -85,B 0,C 180,E1 -10371.034,E2 -10371.034} C_VEL
LIN {X 0,Y 411.222,Z 382.763,A -85,B 0,C 180,E1 -10374.215,E2 -10374.215} C_VEL
LIN {X 0,Y 411.254,Z 382.756,A -85,B 0,C 180,E1 -10377.477,E2 -10377.477} C_VEL
LIN {X 0,Y 411.192,Z 382.762,A -85,B 0,C 180,E1 -10380.847,E2 -10380.847} C_VEL
LIN {X 0,Y 411.2,Z 382.745,A -85,B 0,C 180,E1 -10384.333,E2 -10384.333} C_VEL
LIN {X 0,Y 411.198,Z 382.763,A -85,B 0,C 180,E1 -10387.972,E2 -10387.972} C_VEL
LIN {X 0,Y 411.193,Z 382.735,A -85,B 0,C 180,E1 -10391.234,E2 -10391.234} C_VEL
LIN {X 0,Y 411.17,Z 382.756,A -85,B 0,C 180,E1 -10394.49,E2 -10394.49} C_VEL
LIN {X 0,Y 411.192,Z 382.763,A -85,B 0,C 180,E1 -10398.197,E2 -10398.197} C_VEL
LIN {X 0,Y 411.221,Z 382.76,A -85,B 0,C 180,E1 -10400.777,E2 -10400.777} C_VEL
LIN {X 0,Y 411.192,Z 382.757,A -85,B 0,C 180,E1 -10404.471,E2 -10404.471} C_VEL
LIN {X 0,Y 411.162,Z 382.766,A -85,B 0,C 180,E1 -10408.003,E2 -10408.003} C_VEL
LIN {X 0,Y 411.217,Z 382.75,A -85,B 0,C 180,E1 -10411.411,E2 -10411.411} C_VEL
LIN {X 0,Y 411.229,Z 382.757,A -85,B 0,C 180,E1 -10414.707,E2 -10414.707} C_VEL
LIN {X 0,Y 411.199,Z 382.761,A -85,B 0,C 180,E1 -10417.914,E2 -10417.914} C_VEL
LIN {X 0,Y 411.217,Z 382.743,A -85,B 0,C 180,E1 -10421.052,E2 -10421.052} C_VEL
LIN {X 0,Y 411.248,Z 382.755,A -85,B 0,C 180,E1 -10424.132,E2 -10424.132} C_VEL
LIN {X 0,Y 411.308,Z 382.743,A -85,B 0,C 180,E1 -10427.166,E2 -10427.166} C_VEL
LIN {X 0,Y 411.29,Z 382.73,A -85,B 0,C 180,E1 -10430.162,E2 -10430.162} C_VEL
LIN {X 0,Y 411.454,Z 382.728,A -85,B 0,C 180,E1 -10433.134,E2 -10433.134} C_VEL
LIN {X 0,Y 411.307,Z 382.748,A -85,B 0,C 180,E1 -10435.1,E2 -10435.1} C_VEL
LIN {X 0,Y 411.508,Z 382.713,A -85,B 0,C 180,E1 -10438.043,E2 -10438.043} C_VEL
LIN {X 0,Y 411.636,Z 382.685,A -85,B 0,C 180,E1 -10440.001,E2 -10440.001} C_VEL
LIN {X 0,Y 411.461,Z 382.728,A -85,B 0,C 180,E1 -10442.938,E2 -10442.938} C_VEL
LIN {X 0,Y 411.455,Z 382.722,A -85,B 0,C 180,E1 -10446.868,E2 -10446.868} C_VEL
LIN {X 0,Y 411.288,Z 382.727,A -85,B 0,C 180,E1 -10449.839,E2 -10449.839} C_VEL
LIN {X 0,Y 411.3,Z 382.746,A -85,B 0,C 180,E1 -10453.105,E2 -10453.105} C_VEL
LIN {X 0,Y 411.259,Z 382.741,A -85,B 0,C 180,E1 -10456.87,E2 -10456.87} C_VEL
LIN {X 0,Y 411.226,Z 382.746,A -85,B 0,C 180,E1 -10459.988,E2 -10459.988} C_VEL
LIN {X 0,Y 411.199,Z 382.76,A -85,B 0,C 180,E1 -10463.148,E2 -10463.148} C_VEL
LIN {X 0,Y 411.234,Z 382.742,A -85,B 0,C 180,E1 -10466.382,E2 -10466.382} C_VEL
LIN {X 0,Y 411.208,Z 382.76,A -85,B 0,C 180,E1 -10469.713,E2 -10469.713} C_VEL
LIN {X 0,Y 411.204,Z 382.752,A -85,B 0,C 180,E1 -10473.157,E2 -10473.157} C_VEL
LIN {X 0,Y 411.193,Z 382.764,A -85,B 0,C 180,E1 -10476.554,E2 -10476.554} C_VEL
LIN {X 0,Y 411.225,Z 382.754,A -85,B 0,C 180,E1 -10479.731,E2 -10479.731} C_VEL
LIN {X 0,Y 411.23,Z 382.757,A -85,B 0,C 180,E1 -10483.127,E2 -10483.127} C_VEL
LIN {X 0,Y 411.171,Z 382.769,A -85,B 0,C 180,E1 -10485.881,E2 -10485.881} C_VEL
LIN {X 0,Y 411.162,Z 382.751,A -85,B 0,C 180,E1 -10488.773,E2 -10488.773} C_VEL
LIN {X 0,Y 411.21,Z 382.765,A -85,B 0,C 180,E1 -10491.831,E2 -10491.831} C_VEL
LIN {X 0,Y 411.212,Z 382.76,A -85,B 0,C 180,E1 -10495.122,E2 -10495.122} C_VEL
LIN {X 0,Y 411.172,Z 382.764,A -85,B 0,C 180,E1 -10498.004,E2 -10498.004} C_VEL
LIN {X 0,Y 411.255,Z 382.943,A -85,B 0,C 180,E1 -10500.541,E2 -10500.541} C_VEL
LIN {X 0,Y 413.194,Z 392.97,A -85,B 0,C 180,E1 -10503.482,E2 -10503.482} C_VEL
LIN {X 0,Y 413.748,Z 396.934,A -85,B 0,C 180,E1 -10504.549,E2 -10504.549} C_VEL
LIN {X 0,Y 413.068,Z 407.506,A -85,B 0,C 180,E1 -10507.228,E2 -10507.228} C_VEL
LIN {X 0,Y 412.258,Z 418.554,A -85,B 0,C 180,E1 -10510.066,E2 -10510.066} C_VEL
LIN {X 0,Y 412.157,Z 420.544,A -85,B 0,C 180,E1 -10510.548,E2 -10510.548} C_VEL
LIN {X 0,Y 412.714,Z 423.933,A -85,B 0,C 180,E1 -10510.69,E2 -10510.69} C_VEL
LIN {X 0,Y 416.988,Z 448.083,A -85,B 0,C 180,E1 -10511.324,E2 -10511.324} C_VEL
LIN {X 0,Y 416.138,Z 525.495,A -85,B 0,C 180,E1 -10512.683,E2 -10512.683} C_VEL
LIN {X 0,Y 415.801,Z 535.407,A -85,B 0,C 180,E1 -10512.954,E2 -10512.954} C_VEL
LIN {X 0,Y 415.312,Z 545.392,A -85,B 0,C 180,E1 -10513.345,E2 -10513.345} C_VEL
LIN {X 0,Y 414.77,Z 555.75,A -85,B 0,C 180,E1 -10513.892,E2 -10513.892} C_VEL
LIN {X 0,Y 414.125,Z 564.894,A -85,B 0,C 180,E1 -10514.498,E2 -10514.498} C_VEL
LIN {X 0,Y 413.522,Z 573.898,A -85,B 0,C 180,E1 -10515.231,E2 -10515.231} C_VEL
LIN {X 0,Y 412.879,Z 582.528,A -85,B 0,C 180,E1 -10516.077,E2 -10516.077} C_VEL
LIN {X 0,Y 412.382,Z 590.051,A -85,B 0,C 180,E1 -10516.95,E2 -10516.95} C_VEL
LIN {X 0,Y 411.662,Z 598.848,A -85,B 0,C 180,E1 -10518.179,E2 -10518.179} C_VEL
LIN {X 0,Y 411.159,Z 604.838,A -85,B 0,C 180,E1 -10519.163,E2 -10519.163} C_VEL
LIN {X 0,Y 410.753,Z 611.15,A -85,B 0,C 180,E1 -10520.397,E2 -10520.397} C_VEL
LIN {X 0,Y 410.423,Z 616.424,A -85,B 0,C 180,E1 -10521.631,E2 -10521.631} C_VEL
LIN {X 0,Y 410.169,Z 621.517,A -85,B 0,C 180,E1 -10523.112,E2 -10523.112} C_VEL
LIN {X 0,Y 410.021,Z 625.48,A -85,B 0,C 180,E1 -10524.591,E2 -10524.591} C_VEL
LIN {X 0,Y 409.932,Z 628.411,A -85,B 0,C 180,E1 -10526.068,E2 -10526.068} C_VEL
LIN {X 0,Y 409.926,Z 629.91,A -85,B 0,C 180,E1 -10527.052,E2 -10527.052} C_VEL
LIN {X 0,Y 409.936,Z 631.431,A -85,B 0,C 180,E1 -10529.018,E2 -10529.018} C_VEL
LIN {X 0,Y 409.927,Z 631.709,A -85,B 0,C 180,E1 -10530,E2 -10530} C_VEL
LIN {X 0,Y 409.967,Z 630.837,A -85,B 0,C 180,E1 -10531.965,E2 -10531.965} C_VEL
LIN {X 0,Y 409.926,Z 629.909,A -85,B 0,C 180,E1 -10532.948,E2 -10532.948} C_VEL
LIN {X 0,Y 410.021,Z 626.568,A -85,B 0,C 180,E1 -10534.917,E2 -10534.917} C_VEL
LIN {X 0,Y 410.044,Z 623.44,A -85,B 0,C 180,E1 -10536.224,E2 -10536.224} C_VEL
LIN {X 0,Y 410.207,Z 620.001,A -85,B 0,C 180,E1 -10537.383,E2 -10537.383} C_VEL
LIN {X 0,Y 410.538,Z 614.425,A -85,B 0,C 180,E1 -10538.863,E2 -10538.863} C_VEL
LIN {X 0,Y 410.925,Z 608.772,A -85,B 0,C 180,E1 -10540.097,E2 -10540.097} C_VEL
LIN {X 0,Y 411.385,Z 601.965,A -85,B 0,C 180,E1 -10541.33,E2 -10541.33} C_VEL
LIN {X 0,Y 412.099,Z 593.749,A -85,B 0,C 180,E1 -10542.559,E2 -10542.559} C_VEL
LIN {X 0,Y 412.669,Z 585.919,A -85,B 0,C 180,E1 -10543.543,E2 -10543.543} C_VEL
LIN {X 0,Y 413.257,Z 577.579,A -85,B 0,C 180,E1 -10544.426,E2 -10544.426} C_VEL
LIN {X 0,Y 413.946,Z 568.068,A -85,B 0,C 180,E1 -10545.258,E2 -10545.258} C_VEL
LIN {X 0,Y 414.478,Z 559.676,A -85,B 0,C 180,E1 -10545.868,E2 -10545.868} C_VEL
LIN {X 0,Y 415.133,Z 549.169,A -85,B 0,C 180,E1 -10546.473,E2 -10546.473} C_VEL
LIN {X 0,Y 415.604,Z 538.833,A -85,B 0,C 180,E1 -10546.928,E2 -10546.928} C_VEL
LIN {X 0,Y 416.107,Z 528.114,A -85,B 0,C 180,E1 -10547.255,E2 -10547.255} C_VEL
LIN {X 0,Y 416.424,Z 505.334,A -85,B 0,C 180,E1 -10547.685,E2 -10547.685} C_VEL
LIN {X 0,Y 416.938,Z 447.345,A -85,B 0,C 180,E1 -10548.692,E2 -10548.692} C_VEL
LIN {X 0,Y 412.184,Z 420.814,A -85,B 0,C 180,E1 -10549.419,E2 -10549.419} C_VEL
LIN {X 0,Y 412.206,Z 419.505,A -85,B 0,C 180,E1 -10549.678,E2 -10549.678} C_VEL
LIN {X 0,Y 413.157,Z 406.686,A -85,B 0,C 180,E1 -10553.032,E2 -10553.032} C_VEL
LIN {X 0,Y 413.81,Z 397.154,A -85,B 0,C 180,E1 -10555.46,E2 -10555.46} C_VEL
LIN {X 0,Y 412.718,Z 390.142,A -85,B 0,C 180,E1 -10557.372,E2 -10557.372} C_VEL
LIN {X 0,Y 411.257,Z 382.872,A -85,B 0,C 180,E1 -10559.487,E2 -10559.487} C_VEL
LIN {X 0,Y 411.21,Z 382.758,A -85,B 0,C 180,E1 -10563.155,E2 -10563.155} C_VEL
LIN {X 0,Y 411.198,Z 382.758,A -85,B 0,C 180,E1 -10566.553,E2 -10566.553} C_VEL
LIN {X 0,Y 411.218,Z 382.75,A -85,B 0,C 180,E1 -10569.728,E2 -10569.728} C_VEL
LIN {X 0,Y 411.175,Z 382.764,A -85,B 0,C 180,E1 -10573.133,E2 -10573.133} C_VEL
LIN {X 0,Y 411.238,Z 382.755,A -85,B 0,C 180,E1 -10575.871,E2 -10575.871} C_VEL
LIN {X 0,Y 411.211,Z 382.758,A -85,B 0,C 180,E1 -10578.764,E2 -10578.764} C_VEL
LIN {X 0,Y 411.205,Z 382.765,A -85,B 0,C 180,E1 -10582.027,E2 -10582.027} C_VEL
LIN {X 0,Y 411.207,Z 382.752,A -85,B 0,C 180,E1 -10585.666,E2 -10585.666} C_VEL
LIN {X 0,Y 411.2,Z 382.761,A -85,B 0,C 180,E1 -10589.153,E2 -10589.153} C_VEL
LIN {X 0,Y 411.26,Z 382.739,A -85,B 0,C 180,E1 -10592.522,E2 -10592.522} C_VEL
LIN {X 0,Y 411.227,Z 382.757,A -85,B 0,C 180,E1 -10595.784,E2 -10595.784} C_VEL
LIN {X 0,Y 411.196,Z 382.757,A -85,B 0,C 180,E1 -10598.965,E2 -10598.965} C_VEL
LIN {X 0,Y 411.252,Z 382.739,A -85,B 0,C 180,E1 -10602.084,E2 -10602.084} C_VEL
LIN {X 0,Y 411.263,Z 382.751,A -85,B 0,C 180,E1 -10605.147,E2 -10605.147} C_VEL
LIN {X 0,Y 411.282,Z 382.743,A -85,B 0,C 180,E1 -10608.167,E2 -10608.167} C_VEL
LIN {X 0,Y 411.481,Z 382.717,A -85,B 0,C 180,E1 -10612.146,E2 -10612.146} C_VEL
LIN {X 0,Y 411.473,Z 382.729,A -85,B 0,C 180,E1 -10614.117,E2 -10614.117} C_VEL
LIN {X 0,Y 411.512,Z 382.714,A -85,B 0,C 180,E1 -10618.042,E2 -10618.042} C_VEL
LIN {X 0,Y 411.638,Z 382.684,A -85,B 0,C 180,E1 -10619.999,E2 -10619.999} C_VEL
LIN {X 0,Y 411.464,Z 382.721,A -85,B 0,C 180,E1 -10622.937,E2 -10622.937} C_VEL
LIN {X 0,Y 411.458,Z 382.727,A -85,B 0,C 180,E1 -10626.866,E2 -10626.866} C_VEL
LIN {X 0,Y 411.293,Z 382.73,A -85,B 0,C 180,E1 -10629.838,E2 -10629.838} C_VEL
LIN {X 0,Y 411.311,Z 382.744,A -85,B 0,C 180,E1 -10633.108,E2 -10633.108} C_VEL
LIN {X 0,Y 411.254,Z 382.752,A -85,B 0,C 180,E1 -10636.888,E2 -10636.888} C_VEL
LIN {X 0,Y 411.227,Z 382.746,A -85,B 0,C 180,E1 -10639.986,E2 -10639.986} C_VEL
LIN {X 0,Y 411.2,Z 382.763,A -85,B 0,C 180,E1 -10643.147,E2 -10643.147} C_VEL
LIN {X 0,Y 411.235,Z 382.746,A -85,B 0,C 180,E1 -10646.38,E2 -10646.38} C_VEL
LIN {X 0,Y 411.197,Z 382.765,A -85,B 0,C 180,E1 -10649.712,E2 -10649.712} C_VEL
LIN {X 0,Y 411.203,Z 382.76,A -85,B 0,C 180,E1 -10653.155,E2 -10653.155} C_VEL
LIN {X 0,Y 411.191,Z 382.76,A -85,B 0,C 180,E1 -10656.553,E2 -10656.553} C_VEL
LIN {X 0,Y 411.212,Z 382.754,A -85,B 0,C 180,E1 -10659.728,E2 -10659.728} C_VEL
LIN {X 0,Y 411.174,Z 382.768,A -85,B 0,C 180,E1 -10663.133,E2 -10663.133} C_VEL
LIN {X 0,Y 411.164,Z 382.753,A -85,B 0,C 180,E1 -10665.881,E2 -10665.881} C_VEL
LIN {X 0,Y 411.196,Z 382.734,A -85,B 0,C 180,E1 -10668.766,E2 -10668.766} C_VEL
LIN {X 0,Y 411.201,Z 382.763,A -85,B 0,C 180,E1 -10672.027,E2 -10672.027} C_VEL
LIN {X 0,Y 411.202,Z 382.745,A -85,B 0,C 180,E1 -10675.666,E2 -10675.666} C_VEL
LIN {X 0,Y 411.194,Z 382.762,A -85,B 0,C 180,E1 -10679.153,E2 -10679.153} C_VEL
LIN {X 0,Y 411.256,Z 382.756,A -85,B 0,C 180,E1 -10682.522,E2 -10682.522} C_VEL
LIN {X 0,Y 411.223,Z 382.763,A -85,B 0,C 180,E1 -10685.784,E2 -10685.784} C_VEL
LIN {X 0,Y 411.193,Z 382.768,A -85,B 0,C 180,E1 -10688.966,E2 -10688.966} C_VEL
LIN {X 0,Y 411.249,Z 382.759,A -85,B 0,C 180,E1 -10692.085,E2 -10692.085} C_VEL
LIN {X 0,Y 411.256,Z 382.76,A -85,B 0,C 180,E1 -10695.147,E2 -10695.147} C_VEL
LIN {X 0,Y 411.281,Z 382.756,A -85,B 0,C 180,E1 -10698.167,E2 -10698.167} C_VEL
LIN {X 0,Y 411.478,Z 382.732,A -85,B 0,C 180,E1 -10702.146,E2 -10702.146} C_VEL
LIN {X 0,Y 411.473,Z 382.732,A -85,B 0,C 180,E1 -10704.118,E2 -10704.118} C_VEL
LIN {X 0,Y 411.51,Z 382.727,A -85,B 0,C 180,E1 -10708.042,E2 -10708.042} C_VEL
LIN {X 0,Y 411.639,Z 382.712,A -85,B 0,C 180,E1 -10710,E2 -10710} C_VEL
LIN {X 0,Y 411.463,Z 382.734,A -85,B 0,C 180,E1 -10712.937,E2 -10712.937} C_VEL
LIN {X 0,Y 411.457,Z 382.735,A -85,B 0,C 180,E1 -10716.867,E2 -10716.867} C_VEL
LIN {X 0,Y 411.289,Z 382.754,A -85,B 0,C 180,E1 -10719.838,E2 -10719.838} C_VEL
LIN {X 0,Y 411.278,Z 382.756,A -85,B 0,C 180,E1 -10723.326,E2 -10723.326} C_VEL
LIN {X 0,Y 411.252,Z 382.761,A -85,B 0,C 180,E1 -10726.888,E2 -10726.888} C_VEL
LIN {X 0,Y 411.235,Z 382.76,A -85,B 0,C 180,E1 -10727.592,E2 -10727.592} C_VEL
LIN {X 0,Y 410.575,Z 382.844,A -85,B 0,C 180,E1 -10728.41,E2 -10728.41} C_VEL
LIN {X 0,Y 407.687,Z 383.203,A -85,B 0,C 180,E1 -10729.738,E2 -10729.738} C_VEL
LIN {X 0,Y 405.243,Z 383.509,A -85,B 0,C 180,E1 -10730.811,E2 -10730.811} C_VEL
LIN {X 0,Y 404.207,Z 383.636,A -85,B 0,C 180,E1 -10731.641,E2 -10731.641} C_VEL
LIN {X 0,Y 404.131,Z 383.644,A -85,B 0,C 180,E1 -10731.922,E2 -10731.922} C_VEL
LIN {X 0,Y 404.211,Z 383.637,A -85,B 0,C 180,E1 -10735.296,E2 -10735.296} C_VEL
LIN {X 0,Y 404.192,Z 383.635,A -85,B 0,C 180,E1 -10737.999,E2 -10737.999} C_VEL
LIN {X 0,Y 404.137,Z 383.643,A -85,B 0,C 180,E1 -10741.559,E2 -10741.559} C_VEL
LIN {X 0,Y 404.179,Z 383.619,A -85,B 0,C 180,E1 -10745.016,E2 -10745.016} C_VEL
LIN {X 0,Y 404.157,Z 383.64,A -85,B 0,C 180,E1 -10748.756,E2 -10748.756} C_VEL
LIN {X 0,Y 404.143,Z 383.609,A -85,B 0,C 180,E1 -10751.604,E2 -10751.604} C_VEL
LIN {X 0,Y 404.139,Z 383.632,A -85,B 0,C 180,E1 -10754.522,E2 -10754.522} C_VEL
LIN {X 0,Y 404.166,Z 383.637,A -85,B 0,C 180,E1 -10757.3,E2 -10757.3} C_VEL
LIN {X 0,Y 404.162,Z 383.63,A -85,B 0,C 180,E1 -10759.955,E2 -10759.955} C_VEL
LIN {X 0,Y 404.133,Z 383.641,A -85,B 0,C 180,E1 -10763.124,E2 -10763.124} C_VEL
LIN {X 0,Y 404.138,Z 383.63,A -85,B 0,C 180,E1 -10766.188,E2 -10766.188} C_VEL
LIN {X 0,Y 404.156,Z 383.639,A -85,B 0,C 180,E1 -10769.717,E2 -10769.717} C_VEL
LIN {X 0,Y 404.188,Z 383.624,A -85,B 0,C 180,E1 -10773.123,E2 -10773.123} C_VEL
LIN {X 0,Y 404.17,Z 383.636,A -85,B 0,C 180,E1 -10775.335,E2 -10775.335} C_VEL
LIN {X 0,Y 404.132,Z 383.637,A -85,B 0,C 180,E1 -10778.581,E2 -10778.581} C_VEL
LIN {X 0,Y 404.203,Z 383.617,A -85,B 0,C 180,E1 -10781.762,E2 -10781.762} C_VEL
LIN {X 0,Y 404.201,Z 383.635,A -85,B 0,C 180,E1 -10784.882,E2 -10784.882} C_VEL
LIN {X 0,Y 404.263,Z 383.621,A -85,B 0,C 180,E1 -10787.959,E2 -10787.959} C_VEL
LIN {X 0,Y 404.427,Z 383.596,A -85,B 0,C 180,E1 -10792.1,E2 -10792.1} C_VEL
LIN {X 0,Y 404.418,Z 383.607,A -85,B 0,C 180,E1 -10794.016,E2 -10794.016} C_VEL
LIN {X 0,Y 404.477,Z 383.588,A -85,B 0,C 180,E1 -10798.009,E2 -10798.009} C_VEL
LIN {X 0,Y 404.605,Z 383.56,A -85,B 0,C 180,E1 -10800.001,E2 -10800.001} C_VEL
LIN {X 0,Y 404.418,Z 383.605,A -85,B 0,C 180,E1 -10802.989,E2 -10802.989} C_VEL
LIN {X 0,Y 404.406,Z 383.599,A -85,B 0,C 180,E1 -10806.988,E2 -10806.988} C_VEL
LIN {X 0,Y 404.253,Z 383.604,A -85,B 0,C 180,E1 -10810.012,E2 -10810.012} C_VEL
LIN {X 0,Y 404.261,Z 383.623,A -85,B 0,C 180,E1 -10813.212,E2 -10813.212} C_VEL
LIN {X 0,Y 404.214,Z 383.618,A -85,B 0,C 180,E1 -10817.009,E2 -10817.009} C_VEL
LIN {X 0,Y 404.159,Z 383.631,A -85,B 0,C 180,E1 -10820.352,E2 -10820.352} C_VEL
LIN {X 0,Y 404.166,Z 383.637,A -85,B 0,C 180,E1 -10823.575,E2 -10823.575} C_VEL
LIN {X 0,Y 404.18,Z 383.626,A -85,B 0,C 180,E1 -10825.767,E2 -10825.767} C_VEL
LIN {X 0,Y 404.195,Z 383.624,A -85,B 0,C 180,E1 -10828,E2 -10828} C_VEL
LIN {X 0,Y 404.144,Z 383.641,A -85,B 0,C 180,E1 -10831.561,E2 -10831.561} C_VEL
LIN {X 0,Y 404.183,Z 383.629,A -85,B 0,C 180,E1 -10835.017,E2 -10835.017} C_VEL
LIN {X 0,Y 404.161,Z 383.634,A -85,B 0,C 180,E1 -10838.757,E2 -10838.757} C_VEL
LIN {X 0,Y 404.19,Z 383.635,A -85,B 0,C 180,E1 -10841.612,E2 -10841.612} C_VEL
LIN {X 0,Y 404.191,Z 383.633,A -85,B 0,C 180,E1 -10844.53,E2 -10844.53} C_VEL
LIN {X 0,Y 404.135,Z 383.642,A -85,B 0,C 180,E1 -10847.297,E2 -10847.297} C_VEL
LIN {X 0,Y 404.168,Z 383.624,A -85,B 0,C 180,E1 -10849.956,E2 -10849.956} C_VEL
LIN {X 0,Y 404.14,Z 383.639,A -85,B 0,C 180,E1 -10853.125,E2 -10853.125} C_VEL
LIN {X 0,Y 404.146,Z 383.642,A -85,B 0,C 180,E1 -10856.189,E2 -10856.189} C_VEL
LIN {X 0,Y 404.245,Z 383.742,A -85,B 0,C 180,E1 -10860.222,E2 -10860.222} C_VEL
LIN {X 0,Y 406.171,Z 393.83,A -85,B 0,C 180,E1 -10863.265,E2 -10863.265} C_VEL
LIN {X 0,Y 406.807,Z 399.044,A -85,B 0,C 180,E1 -10864.687,E2 -10864.687} C_VEL
LIN {X 0,Y 405.791,Z 412.508,A -85,B 0,C 180,E1 -10868.139,E2 -10868.139} C_VEL
LIN {X 0,Y 405.191,Z 420.368,A -85,B 0,C 180,E1 -10870.203,E2 -10870.203} C_VEL
LIN {X 0,Y 405.985,Z 424.696,A -85,B 0,C 180,E1 -10870.375,E2 -10870.375} C_VEL
LIN {X 0,Y 410.266,Z 448.806,A -85,B 0,C 180,E1 -10871.023,E2 -10871.023} C_VEL
LIN {X 0,Y 409.37,Z 525.3,A -85,B 0,C 180,E1 -10872.388,E2 -10872.388} C_VEL
LIN {X 0,Y 409.013,Z 535.212,A -85,B 0,C 180,E1 -10872.662,E2 -10872.662} C_VEL
LIN {X 0,Y 408.498,Z 545.197,A -85,B 0,C 180,E1 -10873.059,E2 -10873.059} C_VEL
LIN {X 0,Y 407.954,Z 555.555,A -85,B 0,C 180,E1 -10873.615,E2 -10873.615} C_VEL
LIN {X 0,Y 407.283,Z 564.699,A -85,B 0,C 180,E1 -10874.23,E2 -10874.23} C_VEL
LIN {X 0,Y 406.626,Z 573.702,A -85,B 0,C 180,E1 -10874.975,E2 -10874.975} C_VEL
LIN {X 0,Y 405.964,Z 582.084,A -85,B 0,C 180,E1 -10875.806,E2 -10875.806} C_VEL
LIN {X 0,Y 405.416,Z 589.855,A -85,B 0,C 180,E1 -10876.722,E2 -10876.722} C_VEL
LIN {X 0,Y 404.691,Z 598.652,A -85,B 0,C 180,E1 -10877.972,E2 -10877.972} C_VEL
LIN {X 0,Y 404.153,Z 604.642,A -85,B 0,C 180,E1 -10878.973,E2 -10878.973} C_VEL
LIN {X 0,Y 403.713,Z 610.954,A -85,B 0,C 180,E1 -10880.228,E2 -10880.228} C_VEL
LIN {X 0,Y 403.364,Z 616.228,A -85,B 0,C 180,E1 -10881.484,E2 -10881.484} C_VEL
LIN {X 0,Y 403.082,Z 621.321,A -85,B 0,C 180,E1 -10882.99,E2 -10882.99} C_VEL
LIN {X 0,Y 402.923,Z 625.284,A -85,B 0,C 180,E1 -10884.495,E2 -10884.495} C_VEL
LIN {X 0,Y 402.853,Z 628.216,A -85,B 0,C 180,E1 -10885.999,E2 -10885.999} C_VEL
LIN {X 0,Y 402.824,Z 629.715,A -85,B 0,C 180,E1 -10887,E2 -10887} C_VEL
LIN {X 0,Y 402.863,Z 631.237,A -85,B 0,C 180,E1 -10889.001,E2 -10889.001} C_VEL
LIN {X 0,Y 402.851,Z 631.515,A -85,B 0,C 180,E1 -10890,E2 -10890} C_VEL
LIN {X 0,Y 402.865,Z 630.642,A -85,B 0,C 180,E1 -10892,E2 -10892} C_VEL
LIN {X 0,Y 402.825,Z 629.714,A -85,B 0,C 180,E1 -10893.001,E2 -10893.001} C_VEL
LIN {X 0,Y 402.933,Z 626.372,A -85,B 0,C 180,E1 -10895.003,E2 -10895.003} C_VEL
LIN {X 0,Y 403.006,Z 622.748,A -85,B 0,C 180,E1 -10896.508,E2 -10896.508} C_VEL
LIN {X 0,Y 403.24,Z 618.016,A -85,B 0,C 180,E1 -10898.015,E2 -10898.015} C_VEL
LIN {X 0,Y 403.634,Z 612.044,A -85,B 0,C 180,E1 -10899.521,E2 -10899.521} C_VEL
LIN {X 0,Y 404.046,Z 605.95,A -85,B 0,C 180,E1 -10900.777,E2 -10900.777} C_VEL
LIN {X 0,Y 404.553,Z 600.209,A -85,B 0,C 180,E1 -10901.778,E2 -10901.778} C_VEL
LIN {X 0,Y 405.144,Z 593.553,A -85,B 0,C 180,E1 -10902.778,E2 -10902.778} C_VEL
LIN {X 0,Y 405.752,Z 585.723,A -85,B 0,C 180,E1 -10903.778,E2 -10903.778} C_VEL
LIN {X 0,Y 406.329,Z 578.03,A -85,B 0,C 180,E1 -10904.614,E2 -10904.614} C_VEL
LIN {X 0,Y 407.099,Z 567.873,A -85,B 0,C 180,E1 -10905.521,E2 -10905.521} C_VEL
LIN {X 0,Y 407.668,Z 559.481,A -85,B 0,C 180,E1 -10906.14,E2 -10906.14} C_VEL
LIN {X 0,Y 408.336,Z 548.974,A -85,B 0,C 180,E1 -10906.756,E2 -10906.756} C_VEL
LIN {X 0,Y 408.821,Z 538.638,A -85,B 0,C 180,E1 -10907.218,E2 -10907.218} C_VEL
LIN {X 0,Y 409.323,Z 527.919,A -85,B 0,C 180,E1 -10907.55,E2 -10907.55} C_VEL
LIN {X 0,Y 409.684,Z 505.139,A -85,B 0,C 180,E1 -10907.986,E2 -10907.986} C_VEL
LIN {X 0,Y 410.17,Z 447.851,A -85,B 0,C 180,E1 -10908.999,E2 -10908.999} C_VEL
LIN {X 0,Y 405.241,Z 420.764,A -85,B 0,C 180,E1 -10909.755,E2 -10909.755} C_VEL
LIN {X 0,Y 405.23,Z 419.804,A -85,B 0,C 180,E1 -10909.899,E2 -10909.899} C_VEL
LIN {X 0,Y 406.292,Z 406.162,A -85,B 0,C 180,E1 -10913.538,E2 -10913.538} C_VEL
LIN {X 0,Y 406.849,Z 398.273,A -85,B 0,C 180,E1 -10915.585,E2 -10915.585} C_VEL
LIN {X 0,Y 405.441,Z 389.961,A -85,B 0,C 180,E1 -10917.906,E2 -10917.906} C_VEL
LIN {X 0,Y 404.244,Z 383.75,A -85,B 0,C 180,E1 -10919.755,E2 -10919.755} C_VEL
LIN {X 0,Y 404.174,Z 383.636,A -85,B 0,C 180,E1 -10923.42,E2 -10923.42} C_VEL
LIN {X 0,Y 404.146,Z 383.633,A -85,B 0,C 180,E1 -10926.246,E2 -10926.246} C_VEL
LIN {X 0,Y 404.16,Z 383.638,A -85,B 0,C 180,E1 -10928.756,E2 -10928.756} C_VEL
LIN {X 0,Y 404.124,Z 383.629,A -85,B 0,C 180,E1 -10931.599,E2 -10931.599} C_VEL
LIN {X 0,Y 404.155,Z 383.638,A -85,B 0,C 180,E1 -10934.523,E2 -10934.523} C_VEL
LIN {X 0,Y 404.212,Z 383.632,A -85,B 0,C 180,E1 -10937.305,E2 -10937.305} C_VEL
LIN {X 0,Y 404.17,Z 383.633,A -85,B 0,C 180,E1 -10939.955,E2 -10939.955} C_VEL
LIN {X 0,Y 404.141,Z 383.641,A -85,B 0,C 180,E1 -10943.124,E2 -10943.124} C_VEL
LIN {X 0,Y 404.146,Z 383.63,A -85,B 0,C 180,E1 -10946.187,E2 -10946.187} C_VEL
LIN {X 0,Y 404.155,Z 383.644,A -85,B 0,C 180,E1 -10949.715,E2 -10949.715} C_VEL
LIN {X 0,Y 404.195,Z 383.618,A -85,B 0,C 180,E1 -10953.122,E2 -10953.122} C_VEL
LIN {X 0,Y 404.177,Z 383.63,A -85,B 0,C 180,E1 -10955.334,E2 -10955.334} C_VEL
LIN {X 0,Y 404.138,Z 383.637,A -85,B 0,C 180,E1 -10958.58,E2 -10958.58} C_VEL
LIN {X 0,Y 404.21,Z 383.613,A -85,B 0,C 180,E1 -10961.761,E2 -10961.761} C_VEL
LIN {X 0,Y 404.21,Z 383.628,A -85,B 0,C 180,E1 -10964.882,E2 -10964.882} C_VEL
LIN {X 0,Y 404.255,Z 383.62,A -85,B 0,C 180,E1 -10967.958,E2 -10967.958} C_VEL
LIN {X 0,Y 404.432,Z 383.593,A -85,B 0,C 180,E1 -10972.099,E2 -10972.099} C_VEL
LIN {X 0,Y 404.422,Z 383.608,A -85,B 0,C 180,E1 -10974.014,E2 -10974.014} C_VEL
LIN {X 0,Y 404.481,Z 383.59,A -85,B 0,C 180,E1 -10978.008,E2 -10978.008} C_VEL
LIN {X 0,Y 404.607,Z 383.559,A -85,B 0,C 180,E1 -10979.999,E2 -10979.999} C_VEL
LIN {X 0,Y 404.421,Z 383.598,A -85,B 0,C 180,E1 -10982.988,E2 -10982.988} C_VEL
LIN {X 0,Y 404.409,Z 383.606,A -85,B 0,C 180,E1 -10986.987,E2 -10986.987} C_VEL
LIN {X 0,Y 404.259,Z 383.605,A -85,B 0,C 180,E1 -10990.011,E2 -10990.011} C_VEL
LIN {X 0,Y 404.264,Z 383.623,A -85,B 0,C 180,E1 -10993.211,E2 -10993.211} C_VEL
LIN {X 0,Y 404.213,Z 383.63,A -85,B 0,C 180,E1 -10997.007,E2 -10997.007} C_VEL
LIN {X 0,Y 404.16,Z 383.627,A -85,B 0,C 180,E1 -11000.351,E2 -11000.351} C_VEL
LIN {X 0,Y 404.166,Z 383.642,A -85,B 0,C 180,E1 -11003.574,E2 -11003.574} C_VEL
LIN {X 0,Y 404.18,Z 383.628,A -85,B 0,C 180,E1 -11005.766,E2 -11005.766} C_VEL
LIN {X 0,Y 404.192,Z 383.624,A -85,B 0,C 180,E1 -11007.999,E2 -11007.999} C_VEL
LIN {X 0,Y 404.136,Z 383.645,A -85,B 0,C 180,E1 -11011.558,E2 -11011.558} C_VEL
LIN {X 0,Y 404.181,Z 383.624,A -85,B 0,C 180,E1 -11015.016,E2 -11015.016} C_VEL
LIN {X 0,Y 404.154,Z 383.641,A -85,B 0,C 180,E1 -11018.756,E2 -11018.756} C_VEL
LIN {X 0,Y 404.12,Z 383.641,A -85,B 0,C 180,E1 -11021.6,E2 -11021.6} C_VEL
LIN {X 0,Y 404.145,Z 383.639,A -85,B 0,C 180,E1 -11024.522,E2 -11024.522} C_VEL
LIN {X 0,Y 404.141,Z 383.611,A -85,B 0,C 180,E1 -11027.296,E2 -11027.296} C_VEL
LIN {X 0,Y 404.165,Z 383.629,A -85,B 0,C 180,E1 -11029.955,E2 -11029.955} C_VEL
LIN {X 0,Y 404.137,Z 383.642,A -85,B 0,C 180,E1 -11033.124,E2 -11033.124} C_VEL
LIN {X 0,Y 404.141,Z 383.628,A -85,B 0,C 180,E1 -11036.187,E2 -11036.187} C_VEL
LIN {X 0,Y 404.15,Z 383.632,A -85,B 0,C 180,E1 -11039.715,E2 -11039.715} C_VEL
LIN {X 0,Y 404.192,Z 383.64,A -85,B 0,C 180,E1 -11043.123,E2 -11043.123} C_VEL
LIN {X 0,Y 404.174,Z 383.642,A -85,B 0,C 180,E1 -11045.334,E2 -11045.334} C_VEL
LIN {X 0,Y 404.135,Z 383.646,A -85,B 0,C 180,E1 -11048.58,E2 -11048.58} C_VEL
LIN {X 0,Y 404.207,Z 383.637,A -85,B 0,C 180,E1 -11051.762,E2 -11051.762} C_VEL
LIN {X 0,Y 404.203,Z 383.638,A -85,B 0,C 180,E1 -11054.882,E2 -11054.882} C_VEL
LIN {X 0,Y 404.253,Z 383.631,A -85,B 0,C 180,E1 -11057.958,E2 -11057.958} C_VEL
LIN {X 0,Y 404.43,Z 383.61,A -85,B 0,C 180,E1 -11062.099,E2 -11062.099} C_VEL
LIN {X 0,Y 404.421,Z 383.61,A -85,B 0,C 180,E1 -11064.015,E2 -11064.015} C_VEL
LIN {X 0,Y 404.479,Z 383.603,A -85,B 0,C 180,E1 -11068.008,E2 -11068.008} C_VEL
LIN {X 0,Y 404.608,Z 383.588,A -85,B 0,C 180,E1 -11070,E2 -11070} C_VEL
LIN {X 0,Y 404.42,Z 383.611,A -85,B 0,C 180,E1 -11072.988,E2 -11072.988} C_VEL
LIN {X 0,Y 404.408,Z 383.613,A -85,B 0,C 180,E1 -11076.987,E2 -11076.987} C_VEL
LIN {X 0,Y 404.255,Z 383.631,A -85,B 0,C 180,E1 -11080.011,E2 -11080.011} C_VEL
LIN {X 0,Y 404.262,Z 383.631,A -85,B 0,C 180,E1 -11083.211,E2 -11083.211} C_VEL
LIN {X 0,Y 404.211,Z 383.638,A -85,B 0,C 180,E1 -11087.007,E2 -11087.007} C_VEL
LIN {X 0,Y 404.159,Z 383.643,A -85,B 0,C 180,E1 -11090.351,E2 -11090.351} C_VEL
LIN {X 0,Y 404.131,Z 383.644,A -85,B 0,C 180,E1 -11091.922,E2 -11091.922} C_VEL
LIN {X 0,Y 403.489,Z 383.728,A -85,B 0,C 180,E1 -11092.753,E2 -11092.753} C_VEL
LIN {X 0,Y 400.656,Z 384.084,A -85,B 0,C 180,E1 -11094.105,E2 -11094.105} C_VEL
LIN {X 0,Y 398.246,Z 384.384,A -85,B 0,C 180,E1 -11095.197,E2 -11095.197} C_VEL
LIN {X 0,Y 397.212,Z 384.509,A -85,B 0,C 180,E1 -11096.042,E2 -11096.042} C_VEL
LIN {X 0,Y 397.129,Z 384.517,A -85,B 0,C 180,E1 -11096.328,E2 -11096.328} C_VEL
LIN {X 0,Y 397.121,Z 384.507,A -85,B 0,C 180,E1 -11098.543,E2 -11098.543} C_VEL
LIN {X 0,Y 397.075,Z 384.524,A -85,B 0,C 180,E1 -11102.071,E2 -11102.071} C_VEL
LIN {X 0,Y 397.114,Z 384.503,A -85,B 0,C 180,E1 -11105.503,E2 -11105.503} C_VEL
LIN {X 0,Y 397.131,Z 384.514,A -85,B 0,C 180,E1 -11108.863,E2 -11108.863} C_VEL
LIN {X 0,Y 397.077,Z 384.487,A -85,B 0,C 180,E1 -11112.265,E2 -11112.265} C_VEL
LIN {X 0,Y 397.083,Z 384.519,A -85,B 0,C 180,E1 -11115.068,E2 -11115.068} C_VEL
LIN {X 0,Y 397.103,Z 384.517,A -85,B 0,C 180,E1 -11118.014,E2 -11118.014} C_VEL
LIN {X 0,Y 397.128,Z 384.517,A -85,B 0,C 180,E1 -11121.138,E2 -11121.138} C_VEL
LIN {X 0,Y 397.113,Z 384.509,A -85,B 0,C 180,E1 -11124.497,E2 -11124.497} C_VEL
LIN {X 0,Y 397.074,Z 384.52,A -85,B 0,C 180,E1 -11127.929,E2 -11127.929} C_VEL
LIN {X 0,Y 397.141,Z 384.514,A -85,B 0,C 180,E1 -11130.298,E2 -11130.298} C_VEL
LIN {X 0,Y 397.188,Z 384.493,A -85,B 0,C 180,E1 -11132.61,E2 -11132.61} C_VEL
LIN {X 0,Y 397.126,Z 384.515,A -85,B 0,C 180,E1 -11135.982,E2 -11135.982} C_VEL
LIN {X 0,Y 397.131,Z 384.502,A -85,B 0,C 180,E1 -11139.705,E2 -11139.705} C_VEL
LIN {X 0,Y 397.175,Z 384.505,A -85,B 0,C 180,E1 -11142.845,E2 -11142.845} C_VEL
LIN {X 0,Y 397.22,Z 384.501,A -85,B 0,C 180,E1 -11146.679,E2 -11146.679} C_VEL
LIN {X 0,Y 397.216,Z 384.481,A -85,B 0,C 180,E1 -11149.81,E2 -11149.81} C_VEL
LIN {X 0,Y 397.358,Z 384.485,A -85,B 0,C 180,E1 -11152.889,E2 -11152.889} C_VEL
LIN {X 0,Y 397.25,Z 384.5,A -85,B 0,C 180,E1 -11154.926,E2 -11154.926} C_VEL
LIN {X 0,Y 397.446,Z 384.464,A -85,B 0,C 180,E1 -11157.974,E2 -11157.974} C_VEL
LIN {X 0,Y 397.575,Z 384.434,A -85,B 0,C 180,E1 -11160.001,E2 -11160.001} C_VEL
LIN {X 0,Y 397.377,Z 384.482,A -85,B 0,C 180,E1 -11163.042,E2 -11163.042} C_VEL
LIN {X 0,Y 397.358,Z 384.477,A -85,B 0,C 180,E1 -11167.112,E2 -11167.112} C_VEL
LIN {X 0,Y 397.213,Z 384.482,A -85,B 0,C 180,E1 -11170.192,E2 -11170.192} C_VEL
LIN {X 0,Y 397.222,Z 384.5,A -85,B 0,C 180,E1 -11173.322,E2 -11173.322} C_VEL
LIN {X 0,Y 397.166,Z 384.5,A -85,B 0,C 180,E1 -11176.447,E2 -11176.447} C_VEL
LIN {X 0,Y 397.144,Z 384.496,A -85,B 0,C 180,E1 -11179.648,E2 -11179.648} C_VEL
LIN {X 0,Y 397.131,Z 384.512,A -85,B 0,C 180,E1 -11183.041,E2 -11183.041} C_VEL
LIN {X 0,Y 397.132,Z 384.498,A -85,B 0,C 180,E1 -11186.259,E2 -11186.259} C_VEL
LIN {X 0,Y 397.124,Z 384.513,A -85,B 0,C 180,E1 -11188.544,E2 -11188.544} C_VEL
LIN {X 0,Y 397.109,Z 384.516,A -85,B 0,C 180,E1 -11192.069,E2 -11192.069} C_VEL
LIN {X 0,Y 397.118,Z 384.51,A -85,B 0,C 180,E1 -11195.504,E2 -11195.504} C_VEL
LIN {X 0,Y 397.135,Z 384.508,A -85,B 0,C 180,E1 -11198.864,E2 -11198.864} C_VEL
LIN {X 0,Y 397.159,Z 384.514,A -85,B 0,C 180,E1 -11202.256,E2 -11202.256} C_VEL
LIN {X 0,Y 397.111,Z 384.515,A -85,B 0,C 180,E1 -11205.066,E2 -11205.066} C_VEL
LIN {X 0,Y 397.065,Z 384.513,A -85,B 0,C 180,E1 -11208.022,E2 -11208.022} C_VEL
LIN {X 0,Y 397.132,Z 384.513,A -85,B 0,C 180,E1 -11211.139,E2 -11211.139} C_VEL
LIN {X 0,Y 397.12,Z 384.509,A -85,B 0,C 180,E1 -11214.497,E2 -11214.497} C_VEL
LIN {X 0,Y 397.083,Z 384.518,A -85,B 0,C 180,E1 -11217.93,E2 -11217.93} C_VEL
LIN {X 0,Y 397.194,Z 384.697,A -85,B 0,C 180,E1 -11219.978,E2 -11219.978} C_VEL
LIN {X 0,Y 399.114,Z 394.678,A -85,B 0,C 180,E1 -11223.034,E2 -11223.034} C_VEL
LIN {X 0,Y 399.838,Z 399.906,A -85,B 0,C 180,E1 -11224.493,E2 -11224.493} C_VEL
LIN {X 0,Y 398.955,Z 411.301,A -85,B 0,C 180,E1 -11227.472,E2 -11227.472} C_VEL
LIN {X 0,Y 398.271,Z 420.167,A -85,B 0,C 180,E1 -11229.844,E2 -11229.844} C_VEL
LIN {X 0,Y 399.07,Z 424.494,A -85,B 0,C 180,E1 -11230.02,E2 -11230.02} C_VEL
LIN {X 0,Y 403.503,Z 449.127,A -85,B 0,C 180,E1 -11230.702,E2 -11230.702} C_VEL
LIN {X 0,Y 402.608,Z 525.105,A -85,B 0,C 180,E1 -11232.082,E2 -11232.082} C_VEL
LIN {X 0,Y 402.23,Z 535.017,A -85,B 0,C 180,E1 -11232.36,E2 -11232.36} C_VEL
LIN {X 0,Y 401.716,Z 545.002,A -85,B 0,C 180,E1 -11232.764,E2 -11232.764} C_VEL
LIN {X 0,Y 401.146,Z 555.36,A -85,B 0,C 180,E1 -11233.329,E2 -11233.329} C_VEL
LIN {X 0,Y 400.435,Z 564.504,A -85,B 0,C 180,E1 -11233.953,E2 -11233.953} C_VEL
LIN {X 0,Y 399.732,Z 573.506,A -85,B 0,C 180,E1 -11234.709,E2 -11234.709} C_VEL
LIN {X 0,Y 399.01,Z 582.618,A -85,B 0,C 180,E1 -11235.64,E2 -11235.64} C_VEL
LIN {X 0,Y 398.449,Z 589.794,A -85,B 0,C 180,E1 -11236.504,E2 -11236.504} C_VEL
LIN {X 0,Y 397.729,Z 598.457,A -85,B 0,C 180,E1 -11237.758,E2 -11237.758} C_VEL
LIN {X 0,Y 397.157,Z 604.446,A -85,B 0,C 180,E1 -11238.776,E2 -11238.776} C_VEL
LIN {X 0,Y 396.68,Z 610.758,A -85,B 0,C 180,E1 -11240.053,E2 -11240.053} C_VEL
LIN {X 0,Y 396.322,Z 616.032,A -85,B 0,C 180,E1 -11241.331,E2 -11241.331} C_VEL
LIN {X 0,Y 396.01,Z 621.126,A -85,B 0,C 180,E1 -11242.864,E2 -11242.864} C_VEL
LIN {X 0,Y 395.833,Z 624.643,A -85,B 0,C 180,E1 -11244.188,E2 -11244.188} C_VEL
LIN {X 0,Y 395.776,Z 628.021,A -85,B 0,C 180,E1 -11245.927,E2 -11245.927} C_VEL
LIN {X 0,Y 395.728,Z 629.519,A -85,B 0,C 180,E1 -11246.946,E2 -11246.946} C_VEL
LIN {X 0,Y 395.792,Z 631.042,A -85,B 0,C 180,E1 -11248.983,E2 -11248.983} C_VEL
LIN {X 0,Y 395.779,Z 631.32,A -85,B 0,C 180,E1 -11250,E2 -11250} C_VEL
LIN {X 0,Y 395.763,Z 630.447,A -85,B 0,C 180,E1 -11252.036,E2 -11252.036} C_VEL
LIN {X 0,Y 395.728,Z 629.519,A -85,B 0,C 180,E1 -11253.054,E2 -11253.054} C_VEL
LIN {X 0,Y 395.846,Z 626.177,A -85,B 0,C 180,E1 -11255.093,E2 -11255.093} C_VEL
LIN {X 0,Y 395.922,Z 622.552,A -85,B 0,C 180,E1 -11256.625,E2 -11256.625} C_VEL
LIN {X 0,Y 396.193,Z 617.82,A -85,B 0,C 180,E1 -11258.159,E2 -11258.159} C_VEL
LIN {X 0,Y 396.613,Z 611.849,A -85,B 0,C 180,E1 -11259.692,E2 -11259.692} C_VEL
LIN {X 0,Y 397.036,Z 605.754,A -85,B 0,C 180,E1 -11260.97,E2 -11260.97} C_VEL
LIN {X 0,Y 397.587,Z 600.014,A -85,B 0,C 180,E1 -11261.988,E2 -11261.988} C_VEL
LIN {X 0,Y 398.194,Z 593.357,A -85,B 0,C 180,E1 -11263.005,E2 -11263.005} C_VEL
LIN {X 0,Y 398.841,Z 585.592,A -85,B 0,C 180,E1 -11264.014,E2 -11264.014} C_VEL
LIN {X 0,Y 399.427,Z 577.834,A -85,B 0,C 180,E1 -11264.873,E2 -11264.873} C_VEL
LIN {X 0,Y 400.237,Z 567.678,A -85,B 0,C 180,E1 -11265.794,E2 -11265.794} C_VEL
LIN {X 0,Y 400.851,Z 559.286,A -85,B 0,C 180,E1 -11266.422,E2 -11266.422} C_VEL
LIN {X 0,Y 401.534,Z 548.779,A -85,B 0,C 180,E1 -11267.048,E2 -11267.048} C_VEL
LIN {X 0,Y 402.042,Z 538.443,A -85,B 0,C 180,E1 -11267.518,E2 -11267.518} C_VEL
LIN {X 0,Y 402.548,Z 527.723,A -85,B 0,C 180,E1 -11267.856,E2 -11267.856} C_VEL
LIN {X 0,Y 402.94,Z 504.945,A -85,B 0,C 180,E1 -11268.298,E2 -11268.298} C_VEL
LIN {X 0,Y 403.455,Z 448.855,A -85,B 0,C 180,E1 -11269.306,E2 -11269.306} C_VEL
LIN {X 0,Y 398.324,Z 420.641,A -85,B 0,C 180,E1 -11270.108,E2 -11270.108} C_VEL
LIN {X 0,Y 398.28,Z 419.61,A -85,B 0,C 180,E1 -11270.262,E2 -11270.262} C_VEL
LIN {X 0,Y 399.404,Z 406.331,A -85,B 0,C 180,E1 -11273.873,E2 -11273.873} C_VEL
LIN {X 0,Y 399.866,Z 399.136,A -85,B 0,C 180,E1 -11275.785,E2 -11275.785} C_VEL
LIN {X 0,Y 398.203,Z 389.78,A -85,B 0,C 180,E1 -11278.459,E2 -11278.459} C_VEL
LIN {X 0,Y 397.189,Z 384.621,A -85,B 0,C 180,E1 -11280.06,E2 -11280.06} C_VEL
LIN {X 0,Y 397.122,Z 384.517,A -85,B 0,C 180,E1 -11283.718,E2 -11283.718} C_VEL
LIN {X 0,Y 397.1,Z 384.517,A -85,B 0,C 180,E1 -11287.209,E2 -11287.209} C_VEL
LIN {X 0,Y 397.103,Z 384.5,A -85,B 0,C 180,E1 -11290.445,E2 -11290.445} C_VEL
LIN {X 0,Y 397.104,Z 384.52,A -85,B 0,C 180,E1 -11293.648,E2 -11293.648} C_VEL
LIN {X 0,Y 397.166,Z 384.51,A -85,B 0,C 180,E1 -11296.511,E2 -11296.511} C_VEL
LIN {X 0,Y 397.124,Z 384.512,A -85,B 0,C 180,E1 -11299.55,E2 -11299.55} C_VEL
LIN {X 0,Y 397.099,Z 384.518,A -85,B 0,C 180,E1 -11302.79,E2 -11302.79} C_VEL
LIN {X 0,Y 397.119,Z 384.505,A -85,B 0,C 180,E1 -11306.281,E2 -11306.281} C_VEL
LIN {X 0,Y 397.087,Z 384.519,A -85,B 0,C 180,E1 -11309.118,E2 -11309.118} C_VEL
LIN {X 0,Y 397.195,Z 384.49,A -85,B 0,C 180,E1 -11312.609,E2 -11312.609} C_VEL
LIN {X 0,Y 397.133,Z 384.515,A -85,B 0,C 180,E1 -11315.981,E2 -11315.981} C_VEL
LIN {X 0,Y 397.138,Z 384.504,A -85,B 0,C 180,E1 -11319.704,E2 -11319.704} C_VEL
LIN {X 0,Y 397.183,Z 384.493,A -85,B 0,C 180,E1 -11322.843,E2 -11322.843} C_VEL
LIN {X 0,Y 397.178,Z 384.51,A -85,B 0,C 180,E1 -11325.656,E2 -11325.656} C_VEL
LIN {X 0,Y 397.197,Z 384.494,A -85,B 0,C 180,E1 -11328.776,E2 -11328.776} C_VEL
LIN {X 0,Y 397.394,Z 384.467,A -85,B 0,C 180,E1 -11332.04,E2 -11332.04} C_VEL
LIN {X 0,Y 397.253,Z 384.498,A -85,B 0,C 180,E1 -11334.925,E2 -11334.925} C_VEL
LIN {X 0,Y 397.45,Z 384.466,A -85,B 0,C 180,E1 -11337.973,E2 -11337.973} C_VEL
LIN {X 0,Y 397.576,Z 384.434,A -85,B 0,C 180,E1 -11339.999,E2 -11339.999} C_VEL
LIN {X 0,Y 397.38,Z 384.476,A -85,B 0,C 180,E1 -11343.041,E2 -11343.041} C_VEL
LIN {X 0,Y 397.362,Z 384.485,A -85,B 0,C 180,E1 -11347.111,E2 -11347.111} C_VEL
LIN {X 0,Y 397.219,Z 384.481,A -85,B 0,C 180,E1 -11350.19,E2 -11350.19} C_VEL
LIN {X 0,Y 397.224,Z 384.501,A -85,B 0,C 180,E1 -11353.321,E2 -11353.321} C_VEL
LIN {X 0,Y 397.179,Z 384.505,A -85,B 0,C 180,E1 -11357.155,E2 -11357.155} C_VEL
LIN {X 0,Y 397.099,Z 384.506,A -85,B 0,C 180,E1 -11360.729,E2 -11360.729} C_VEL
LIN {X 0,Y 397.129,Z 384.514,A -85,B 0,C 180,E1 -11364.018,E2 -11364.018} C_VEL
LIN {X 0,Y 397.191,Z 384.493,A -85,B 0,C 180,E1 -11367.39,E2 -11367.39} C_VEL
LIN {X 0,Y 397.075,Z 384.522,A -85,B 0,C 180,E1 -11370.882,E2 -11370.882} C_VEL
LIN {X 0,Y 397.122,Z 384.501,A -85,B 0,C 180,E1 -11374.493,E2 -11374.493} C_VEL
LIN {X 0,Y 397.102,Z 384.518,A -85,B 0,C 180,E1 -11378.274,E2 -11378.274} C_VEL
LIN {X 0,Y 397.085,Z 384.511,A -85,B 0,C 180,E1 -11380.908,E2 -11380.908} C_VEL
LIN {X 0,Y 397.1,Z 384.52,A -85,B 0,C 180,E1 -11383.648,E2 -11383.648} C_VEL
LIN {X 0,Y 397.1,Z 384.499,A -85,B 0,C 180,E1 -11386.52,E2 -11386.52} C_VEL
LIN {X 0,Y 397.116,Z 384.496,A -85,B 0,C 180,E1 -11389.551,E2 -11389.551} C_VEL
LIN {X 0,Y 397.119,Z 384.519,A -85,B 0,C 180,E1 -11392.785,E2 -11392.785} C_VEL
LIN {X 0,Y 397.115,Z 384.503,A -85,B 0,C 180,E1 -11396.282,E2 -11396.282} C_VEL
LIN {X 0,Y 397.11,Z 384.506,A -85,B 0,C 180,E1 -11400.133,E2 -11400.133} C_VEL
LIN {X 0,Y 397.191,Z 384.509,A -85,B 0,C 180,E1 -11402.61,E2 -11402.61} C_VEL
LIN {X 0,Y 397.129,Z 384.518,A -85,B 0,C 180,E1 -11405.982,E2 -11405.982} C_VEL
LIN {X 0,Y 397.135,Z 384.518,A -85,B 0,C 180,E1 -11409.704,E2 -11409.704} C_VEL
LIN {X 0,Y 397.178,Z 384.513,A -85,B 0,C 180,E1 -11412.845,E2 -11412.845} C_VEL
LIN {X 0,Y 397.225,Z 384.507,A -85,B 0,C 180,E1 -11416.702,E2 -11416.702} C_VEL
LIN {X 0,Y 397.215,Z 384.509,A -85,B 0,C 180,E1 -11419.809,E2 -11419.809} C_VEL
LIN {X 0,Y 397.361,Z 384.491,A -85,B 0,C 180,E1 -11422.888,E2 -11422.888} C_VEL
LIN {X 0,Y 397.253,Z 384.504,A -85,B 0,C 180,E1 -11424.925,E2 -11424.925} C_VEL
LIN {X 0,Y 397.46,Z 384.769,A -85,B 0,C 180,E1 -11428.226,E2 -11428.226} C_VEL
LIN {X 0,Y 397.65,Z 384.874,A -85,B 0,C 180,E1 -11430,E2 -11430} C_VEL
LIN {X 0,Y 397.378,Z 384.566,A -85,B 0,C 180,E1 -11433.041,E2 -11433.041} C_VEL
LIN {X 0,Y 397.36,Z 384.491,A -85,B 0,C 180,E1 -11437.111,E2 -11437.111} C_VEL
LIN {X 0,Y 397.214,Z 384.509,A -85,B 0,C 180,E1 -11440.191,E2 -11440.191} C_VEL
LIN {X 0,Y 397.222,Z 384.508,A -85,B 0,C 180,E1 -11443.321,E2 -11443.321} C_VEL
LIN {X 0,Y 397.177,Z 384.513,A -85,B 0,C 180,E1 -11447.155,E2 -11447.155} C_VEL
LIN {X 0,Y 397.098,Z 384.524,A -85,B 0,C 180,E1 -11450.73,E2 -11450.73} C_VEL
LIN {X 0,Y 397.128,Z 384.518,A -85,B 0,C 180,E1 -11454.018,E2 -11454.018} C_VEL
LIN {X 0,Y 397.129,Z 384.517,A -85,B 0,C 180,E1 -11456.328,E2 -11456.328} C_VEL
LIN {X 0,Y 396.46,Z 384.602,A -85,B 0,C 180,E1 -11457.174,E2 -11457.174} C_VEL
LIN {X 0,Y 393.587,Z 384.946,A -85,B 0,C 180,E1 -11458.55,E2 -11458.55} C_VEL
LIN {X 0,Y 391.15,Z 385.248,A -85,B 0,C 180,E1 -11459.661,E2 -11459.661} C_VEL
LIN {X 0,Y 390.099,Z 385.384,A -85,B 0,C 180,E1 -11460.521,E2 -11460.521} C_VEL
LIN {X 0,Y 390.01,Z 385.395,A -85,B 0,C 180,E1 -11460.813,E2 -11460.813} C_VEL
LIN {X 0,Y 390.062,Z 385.377,A -85,B 0,C 180,E1 -11464.024,E2 -11464.024} C_VEL
LIN {X 0,Y 390.054,Z 385.398,A -85,B 0,C 180,E1 -11467.554,E2 -11467.554} C_VEL
LIN {X 0,Y 390.07,Z 385.367,A -85,B 0,C 180,E1 -11470.825,E2 -11470.825} C_VEL
LIN {X 0,Y 390.049,Z 385.381,A -85,B 0,C 180,E1 -11473.886,E2 -11473.886} C_VEL
LIN {X 0,Y 390.075,Z 385.391,A -85,B 0,C 180,E1 -11477.619,E2 -11477.619} C_VEL
LIN {X 0,Y 390.087,Z 385.394,A -85,B 0,C 180,E1 -11480.908,E2 -11480.908} C_VEL
LIN {X 0,Y 390.078,Z 385.381,A -85,B 0,C 180,E1 -11484.793,E2 -11484.793} C_VEL
LIN {X 0,Y 390.023,Z 385.404,A -85,B 0,C 180,E1 -11488.496,E2 -11488.496} C_VEL
LIN {X 0,Y 390.11,Z 385.376,A -85,B 0,C 180,E1 -11492.07,E2 -11492.07} C_VEL
LIN {X 0,Y 390.073,Z 385.392,A -85,B 0,C 180,E1 -11495.52,E2 -11495.52} C_VEL
LIN {X 0,Y 390.049,Z 385.387,A -85,B 0,C 180,E1 -11498.878,E2 -11498.878} C_VEL
LIN {X 0,Y 390.121,Z 385.373,A -85,B 0,C 180,E1 -11502.167,E2 -11502.167} C_VEL
LIN {X 0,Y 390.14,Z 385.385,A -85,B 0,C 180,E1 -11505.393,E2 -11505.393} C_VEL
LIN {X 0,Y 390.151,Z 385.367,A -85,B 0,C 180,E1 -11508.572,E2 -11508.572} C_VEL
LIN {X 0,Y 390.338,Z 385.349,A -85,B 0,C 180,E1 -11511.994,E2 -11511.994} C_VEL
LIN {X 0,Y 390.222,Z 385.376,A -85,B 0,C 180,E1 -11514.834,E2 -11514.834} C_VEL
LIN {X 0,Y 390.415,Z 385.339,A -85,B 0,C 180,E1 -11517.937,E2 -11517.937} C_VEL
LIN {X 0,Y 390.544,Z 385.309,A -85,B 0,C 180,E1 -11520.001,E2 -11520.001} C_VEL
LIN {X 0,Y 390.311,Z 385.362,A -85,B 0,C 180,E1 -11523.097,E2 -11523.097} C_VEL
LIN {X 0,Y 390.325,Z 385.361,A -85,B 0,C 180,E1 -11526.203,E2 -11526.203} C_VEL
LIN {X 0,Y 390.309,Z 385.344,A -85,B 0,C 180,E1 -11528.283,E2 -11528.283} C_VEL
LIN {X 0,Y 390.166,Z 385.381,A -85,B 0,C 180,E1 -11532.484,E2 -11532.484} C_VEL
LIN {X 0,Y 390.139,Z 385.382,A -85,B 0,C 180,E1 -11535.677,E2 -11535.677} C_VEL
LIN {X 0,Y 390.101,Z 385.37,A -85,B 0,C 180,E1 -11538.923,E2 -11538.923} C_VEL
LIN {X 0,Y 390.036,Z 385.401,A -85,B 0,C 180,E1 -11542.235,E2 -11542.235} C_VEL
LIN {X 0,Y 390.116,Z 385.377,A -85,B 0,C 180,E1 -11545.744,E2 -11545.744} C_VEL
LIN {X 0,Y 390.063,Z 385.392,A -85,B 0,C 180,E1 -11549.11,E2 -11549.11} C_VEL
LIN {X 0,Y 390.053,Z 385.387,A -85,B 0,C 180,E1 -11552.721,E2 -11552.721} C_VEL
LIN {X 0,Y 390.055,Z 385.392,A -85,B 0,C 180,E1 -11555.827,E2 -11555.827} C_VEL
LIN {X 0,Y 390.072,Z 385.388,A -85,B 0,C 180,E1 -11559.22,E2 -11559.22} C_VEL
LIN {X 0,Y 390.121,Z 385.39,A -85,B 0,C 180,E1 -11562.388,E2 -11562.388} C_VEL
LIN {X 0,Y 390.061,Z 385.394,A -85,B 0,C 180,E1 -11565.358,E2 -11565.358} C_VEL
LIN {X 0,Y 390.03,Z 385.387,A -85,B 0,C 180,E1 -11568.188,E2 -11568.188} C_VEL
